gfCNCPoint5[13257] = {X 214.8514, Y 66.0622, Z -7.1667, A 0.000, B 0.000, C 0.000 }
gfCNCPoint5[13258] = {X 213.6675, Y 65.7094, Z -7.1667, A 0.000, B 0.000, C 0.000 }
gfCNCPoint5[13259] = {X 212.5602, Y 65.1615, Z -7.1667, A 0.000, B 0.000, C 0.000 }
gfCNCPoint5[13260] = {X 211.5615, Y 64.4343, Z -7.1667, A 0.000, B 0.000, C 0.000 }
gfCNCPoint5[13261] = {X 210.7002, Y 63.5486, Z -7.1667, A 0.000, B 0.000, C 0.000 }
gfCNCPoint5[13262] = {X 210.0010, Y 62.5301, Z -7.1667, A 0.000, B 0.000, C 0.000 }
gfCNCPoint5[13263] = {X 209.4841, Y 61.4080, Z -7.1667, A 0.000, B 0.000, C 0.000 }
gfCNCPoint5[13264] = {X 209.1643, Y 60.2147, Z -7.1667, A 0.000, B 0.000, C 0.000 }
gfCNCPoint5[13265] = {X 209.0510, Y 58.9845, Z -7.1667, A 0.000, B 0.000, C 0.000 }
gfCNCPoint5[13266] = {X 209.0508, Y 58.0000, Z -7.1667, A 0.000, B 0.000, C 0.000 }
gfCNCPoint5[13267] = {X 209.1477, Y 56.8162, Z -7.1667, A 0.000, B 0.000, C 0.000 }
gfCNCPoint5[13268] = {X 209.4358, Y 55.6638, Z -7.1667, A 0.000, B 0.000, C 0.000 }
gfCNCPoint5[13269] = {X 209.9075, Y 54.5737, Z -7.1667, A 0.000, B 0.000, C 0.000 }
gfCNCPoint5[13270] = {X 210.5502, Y 53.5748, Z -7.1667, A 0.000, B 0.000, C 0.000 }
gfCNCPoint5[13271] = {X 211.3467, Y 52.6937, Z -7.1667, A 0.000, B 0.000, C 0.000 }
gfCNCPoint5[13272] = {X 212.2759, Y 51.9538, Z -7.1667, A 0.000, B 0.000, C 0.000 }
gfCNCPoint5[13273] = {X 213.3131, Y 51.3749, Z -7.1667, A 0.000, B 0.000, C 0.000 }
gfCNCPoint5[13274] = {X 214.4306, Y 50.9724, Z -7.1667, A 0.000, B 0.000, C 0.000 }
gfCNCPoint5[13275] = {X 215.3724, Y 50.7834, Z -7.1667, A 0.000, B 0.000, C 0.000 }
gfCNCPoint5[13276] = {X 216.3308, Y 50.7200, Z -7.1667, A 0.000, B 0.000, C 0.000 }
gfCNCPoint5[13277] = {X 237.2617, Y 50.7200, Z -7.1667, A 0.000, B 0.000, C 0.000 }
gfCNCPoint5[13278] = {X 238.3057, Y 50.7953, Z -7.1667, A 0.000, B 0.000, C 0.000 }
gfCNCPoint5[13279] = {X 239.3282, Y 51.0195, Z -7.1667, A 0.000, B 0.000, C 0.000 }
gfCNCPoint5[13280] = {X 240.3080, Y 51.3880, Z -7.1667, A 0.000, B 0.000, C 0.000 }
gfCNCPoint5[13281] = {X 241.2247, Y 51.8932, Z -7.1667, A 0.000, B 0.000, C 0.000 }
gfCNCPoint5[13282] = {X 242.0740, Y 52.5374, Z -7.1667, A 0.000, B 0.000, C 0.000 }
gfCNCPoint5[13283] = {X 242.8201, Y 53.2987, Z -7.1667, A 0.000, B 0.000, C 0.000 }
gfCNCPoint5[13284] = {X 243.4471, Y 54.1608, Z -7.1667, A 0.000, B 0.000, C 0.000 }
gfCNCPoint5[13285] = {X 243.9414, Y 55.1053, Z -7.1667, A 0.000, B 0.000, C 0.000 }
gfCNCPoint5[13286] = {X 244.2925, Y 56.1117, Z -7.1667, A 0.000, B 0.000, C 0.000 }
gfCNCPoint5[13287] = {X 249.2045, Y 58.0272, Z -7.1667, A 0.000, B 0.000, C 0.000 }
gfCNCPoint5[13288] = {X 272.6717, Y 67.3417, Z -7.1667, A 0.000, B 0.000, C 0.000 }
gfCNCPoint5[13289] = {X 272.6716, Y 65.2836, Z -7.1667, A 0.000, B 0.000, C 0.000 }
gfCNCPoint5[13290] = {X 271.6643, Y 64.6022, Z -7.1667, A 0.000, B 0.000, C 0.000 }
gfCNCPoint5[13291] = {X 270.7845, Y 63.7626, Z -7.1667, A 0.000, B 0.000, C 0.000 }
gfCNCPoint5[13292] = {X 270.0567, Y 62.7883, Z -7.1667, A 0.000, B 0.000, C 0.000 }
gfCNCPoint5[13293] = {X 269.5012, Y 61.7064, Z -7.1667, A 0.000, B 0.000, C 0.000 }
gfCNCPoint5[13294] = {X 269.2026, Y 60.8250, Z -7.1667, A 0.000, B 0.000, C 0.000 }
gfCNCPoint5[13295] = {X 269.0188, Y 59.9127, Z -7.1667, A 0.000, B 0.000, C 0.000 }
gfCNCPoint5[13296] = {X 268.9529, Y 58.9845, Z -7.1667, A 0.000, B 0.000, C 0.000 }
gfCNCPoint5[13297] = {X 268.9527, Y 58.0000, Z -7.1667, A 0.000, B 0.000, C 0.000 }
gfCNCPoint5[13298] = {X 269.0633, Y 56.7358, Z -7.1667, A 0.000, B 0.000, C 0.000 }
gfCNCPoint5[13299] = {X 269.3917, Y 55.5101, Z -7.1667, A 0.000, B 0.000, C 0.000 }
gfCNCPoint5[13300] = {X 269.9280, Y 54.3600, Z -7.1667, A 0.000, B 0.000, C 0.000 }
gfCNCPoint5[13301] = {X 270.6559, Y 53.3205, Z -7.1667, A 0.000, B 0.000, C 0.000 }
gfCNCPoint5[13302] = {X 271.5532, Y 52.4232, Z -7.1667, A 0.000, B 0.000, C 0.000 }
gfCNCPoint5[13303] = {X 272.5927, Y 51.6953, Z -7.1667, A 0.000, B 0.000, C 0.000 }
gfCNCPoint5[13304] = {X 273.7428, Y 51.1590, Z -7.1667, A 0.000, B 0.000, C 0.000 }
gfCNCPoint5[13305] = {X 274.9685, Y 50.8306, Z -7.1667, A 0.000, B 0.000, C 0.000 }
gfCNCPoint5[13306] = {X 276.2327, Y 50.7200, Z -7.1667, A 0.000, B 0.000, C 0.000 }
gfCNCPoint5[13307] = {X 292.7731, Y 50.7200, Z -7.1667, A 0.000, B 0.000, C 0.000 }
gfCNCPoint5[13308] = {X 293.4209, Y 50.7489, Z -7.1667, A 0.000, B 0.000, C 0.000 }
gfCNCPoint5[13309] = {X 294.0636, Y 50.8353, Z -7.1667, A 0.000, B 0.000, C 0.000 }
gfCNCPoint5[13310] = {X 294.7292, Y 50.9877, Z -7.1667, A 0.000, B 0.000, C 0.000 }
gfCNCPoint5[13311] = {X 295.3777, Y 51.2019, Z -7.1667, A 0.000, B 0.000, C 0.000 }
gfCNCPoint5[13312] = {X 298.3089, Y 43.5511, Z -7.1667, A 0.000, B 0.000, C 0.000 }
gfCNCPoint5[13313] = {X 298.4820, Y 42.5283, Z -7.1667, A 0.000, B 0.000, C 0.000 }
gfCNCPoint5[13314] = {X 298.7923, Y 41.5385, Z -7.1667, A 0.000, B 0.000, C 0.000 }
gfCNCPoint5[13315] = {X 299.2339, Y 40.5998, Z -7.1667, A 0.000, B 0.000, C 0.000 }
gfCNCPoint5[13316] = {X 299.7987, Y 39.7298, Z -7.1667, A 0.000, B 0.000, C 0.000 }
gfCNCPoint5[13317] = {X 299.7987, Y 36.9943, Z -7.1667, A 0.000, B 0.000, C 0.000 }
gfCNCPoint5[13318] = {X 296.8149, Y 36.9943, Z -7.1667, A 0.000, B 0.000, C 0.000 }
gfCNCPoint5[13319] = {X 296.8147, Y 39.7480, Z -7.1667, A 0.000, B 0.000, C 0.000 }
gfCNCPoint5[13320] = {X 297.3857, Y 40.6103, Z -7.1667, A 0.000, B 0.000, C 0.000 }
gfCNCPoint5[13321] = {X 297.8305, Y 41.5440, Z -7.1667, A 0.000, B 0.000, C 0.000 }
gfCNCPoint5[13322] = {X 298.1402, Y 42.5307, Z -7.1667, A 0.000, B 0.000, C 0.000 }
gfCNCPoint5[13323] = {X 298.3089, Y 43.5511, Z -7.1667, A 0.000, B 0.000, C 0.000 }
gfCNCPoint5[13324] = {X 296.2363, Y 48.9607, Z -7.1667, A 0.000, B 0.000, C 0.000 }
gfCNCPoint5[13325] = {X 296.6124, Y 49.1139, Z -7.1667, A 0.000, B 0.000, C 0.000 }
gfCNCPoint5[13326] = {X 296.9817, Y 49.2828, Z -7.1667, A 0.000, B 0.000, C 0.000 }
gfCNCPoint5[13327] = {X 297.2571, Y 49.4212, Z -7.1667, A 0.000, B 0.000, C 0.000 }
gfCNCPoint5[13328] = {X 297.5280, Y 49.5683, Z -7.1667, A 0.000, B 0.000, C 0.000 }
gfCNCPoint5[13329] = {X 298.7174, Y 50.3602, Z -7.1667, A 0.000, B 0.000, C 0.000 }
gfCNCPoint5[13330] = {X 299.7774, Y 51.3185, Z -7.1667, A 0.000, B 0.000, C 0.000 }
gfCNCPoint5[13331] = {X 300.6847, Y 52.4224, Z -7.1667, A 0.000, B 0.000, C 0.000 }
gfCNCPoint5[13332] = {X 301.5914, Y 51.3191, Z -7.1667, A 0.000, B 0.000, C 0.000 }
gfCNCPoint5[13333] = {X 302.6506, Y 50.3611, Z -7.1667, A 0.000, B 0.000, C 0.000 }
gfCNCPoint5[13334] = {X 303.8393, Y 49.5695, Z -7.1667, A 0.000, B 0.000, C 0.000 }
gfCNCPoint5[13335] = {X 302.8989, Y 49.0956, Z -7.1667, A 0.000, B 0.000, C 0.000 }
gfCNCPoint5[13336] = {X 302.0820, Y 48.4310, Z -7.1667, A 0.000, B 0.000, C 0.000 }
gfCNCPoint5[13337] = {X 301.4268, Y 47.6067, Z -7.1667, A 0.000, B 0.000, C 0.000 }
gfCNCPoint5[13338] = {X 300.9636, Y 46.6610, Z -7.1667, A 0.000, B 0.000, C 0.000 }
gfCNCPoint5[13339] = {X 300.7923, Y 46.0759, Z -7.1667, A 0.000, B 0.000, C 0.000 }
gfCNCPoint5[13340] = {X 300.6953, Y 45.4741, Z -7.1667, A 0.000, B 0.000, C 0.000 }
gfCNCPoint5[13341] = {X 300.6790, Y 45.2570, Z -7.1667, A 0.000, B 0.000, C 0.000 }
gfCNCPoint5[13342] = {X 300.6724, Y 45.0393, Z -7.1667, A 0.000, B 0.000, C 0.000 }
gfCNCPoint5[13343] = {X 300.6725, Y 44.1884, Z -7.1667, A 0.000, B 0.000, C 0.000 }
gfCNCPoint5[13344] = {X 300.6810, Y 43.9888, Z -7.1667, A 0.000, B 0.000, C 0.000 }
gfCNCPoint5[13345] = {X 300.6970, Y 43.7898, Z -7.1667, A 0.000, B 0.000, C 0.000 }
gfCNCPoint5[13346] = {X 300.8617, Y 42.9110, Z -7.1667, A 0.000, B 0.000, C 0.000 }
gfCNCPoint5[13347] = {X 301.1736, Y 42.0731, Z -7.1667, A 0.000, B 0.000, C 0.000 }
gfCNCPoint5[13348] = {X 301.6237, Y 41.3006, Z -7.1667, A 0.000, B 0.000, C 0.000 }
gfCNCPoint5[13349] = {X 302.1987, Y 40.6160, Z -7.1667, A 0.000, B 0.000, C 0.000 }
gfCNCPoint5[13350] = {X 302.1987, Y 34.5943, Z -7.1667, A 0.000, B 0.000, C 0.000 }
gfCNCPoint5[13351] = {X 294.4151, Y 34.5943, Z -7.1667, A 0.000, B 0.000, C 0.000 }
gfCNCPoint5[13352] = {X 294.4146, Y 40.6550, Z -7.1667, A 0.000, B 0.000, C 0.000 }
gfCNCPoint5[13353] = {X 294.9946, Y 41.3214, Z -7.1667, A 0.000, B 0.000, C 0.000 }
gfCNCPoint5[13354] = {X 295.4475, Y 42.0800, Z -7.1667, A 0.000, B 0.000, C 0.000 }
gfCNCPoint5[13355] = {X 295.7590, Y 42.9067, Z -7.1667, A 0.000, B 0.000, C 0.000 }
gfCNCPoint5[13356] = {X 295.9194, Y 43.7755, Z -7.1667, A 0.000, B 0.000, C 0.000 }
gfCNCPoint5[13357] = {X 295.9350, Y 43.9919, Z -7.1667, A 0.000, B 0.000, C 0.000 }
gfCNCPoint5[13358] = {X 295.9411, Y 44.2089, Z -7.1667, A 0.000, B 0.000, C 0.000 }
gfCNCPoint5[13359] = {X 295.9411, Y 45.0000, Z -7.1667, A 0.000, B 0.000, C 0.000 }
gfCNCPoint5[13360] = {X 295.9354, Y 45.2373, Z -7.1667, A 0.000, B 0.000, C 0.000 }
gfCNCPoint5[13361] = {X 295.9181, Y 45.4741, Z -7.1667, A 0.000, B 0.000, C 0.000 }
gfCNCPoint5[13362] = {X 298.3067, Y 45.7073, Z -7.1667, A 0.000, B 0.000, C 0.000 }
gfCNCPoint5[13363] = {X 298.2010, Y 46.4214, Z -7.1667, A 0.000, B 0.000, C 0.000 }
gfCNCPoint5[13364] = {X 298.0252, Y 47.1215, Z -7.1667, A 0.000, B 0.000, C 0.000 }
gfCNCPoint5[13365] = {X 298.3689, Y 47.2942, Z -7.1667, A 0.000, B 0.000, C 0.000 }
gfCNCPoint5[13366] = {X 298.7069, Y 47.4778, Z -7.1667, A 0.000, B 0.000, C 0.000 }
gfCNCPoint5[13367] = {X 298.4514, Y 46.6051, Z -7.1667, A 0.000, B 0.000, C 0.000 }
gfCNCPoint5[13368] = {X 298.3067, Y 45.7073, Z -7.1667, A 0.000, B 0.000, C 0.000 }
gfCNCPoint5[13369] = {X 295.9181, Y 45.4741, Z -7.1667, A 0.000, B 0.000, C 0.000 }
gfCNCPoint5[13370] = {X 295.8472, Y 45.9528, Z -7.1667, A 0.000, B 0.000, C 0.000 }
gfCNCPoint5[13371] = {X 295.7293, Y 46.4221, Z -7.1667, A 0.000, B 0.000, C 0.000 }
gfCNCPoint5[13372] = {X 295.4314, Y 47.1714, Z -7.1667, A 0.000, B 0.000, C 0.000 }
gfCNCPoint5[13373] = {X 295.0142, Y 47.8614, Z -7.1667, A 0.000, B 0.000, C 0.000 }
gfCNCPoint5[13374] = {X 294.4890, Y 48.4733, Z -7.1667, A 0.000, B 0.000, C 0.000 }
gfCNCPoint5[13375] = {X 295.3741, Y 48.6760, Z -7.1667, A 0.000, B 0.000, C 0.000 }
gfCNCPoint5[13376] = {X 296.2363, Y 48.9607, Z -7.1667, A 0.000, B 0.000, C 0.000 }
gfCNCPoint5[13377] = {X 295.3777, Y 51.2019, Z -7.1667, A 0.000, B 0.000, C 0.000 }
gfCNCPoint5[13378] = {X 296.3498, Y 51.6592, Z -7.1667, A 0.000, B 0.000, C 0.000 }
gfCNCPoint5[13379] = {X 297.2441, Y 52.2547, Z -7.1667, A 0.000, B 0.000, C 0.000 }
gfCNCPoint5[13380] = {X 298.0410, Y 52.9753, Z -7.1667, A 0.000, B 0.000, C 0.000 }
gfCNCPoint5[13381] = {X 298.7231, Y 53.8053, Z -7.1667, A 0.000, B 0.000, C 0.000 }
gfCNCPoint5[13382] = {X 299.2946, Y 54.7645, Z -7.1667, A 0.000, B 0.000, C 0.000 }
gfCNCPoint5[13383] = {X 299.7126, Y 55.7997, Z -7.1667, A 0.000, B 0.000, C 0.000 }
gfCNCPoint5[13384] = {X 299.9675, Y 56.8868, Z -7.1667, A 0.000, B 0.000, C 0.000 }
gfCNCPoint5[13385] = {X 300.0531, Y 58.0000, Z -7.1667, A 0.000, B 0.000, C 0.000 }
gfCNCPoint5[13386] = {X 300.0531, Y 58.9431, Z -7.1667, A 0.000, B 0.000, C 0.000 }
gfCNCPoint5[13387] = {X 299.9650, Y 60.0533, Z -7.1667, A 0.000, B 0.000, C 0.000 }
gfCNCPoint5[13388] = {X 299.7090, Y 61.1372, Z -7.1667, A 0.000, B 0.000, C 0.000 }
gfCNCPoint5[13389] = {X 299.2910, Y 62.1695, Z -7.1667, A 0.000, B 0.000, C 0.000 }
gfCNCPoint5[13390] = {X 298.7208, Y 63.1261, Z -7.1667, A 0.000, B 0.000, C 0.000 }
gfCNCPoint5[13391] = {X 300.6826, Y 64.5087, Z -7.1667, A 0.000, B 0.000, C 0.000 }
gfCNCPoint5[13392] = {X 299.7833, Y 65.6047, Z -7.1667, A 0.000, B 0.000, C 0.000 }
gfCNCPoint5[13393] = {X 298.7338, Y 66.5579, Z -7.1667, A 0.000, B 0.000, C 0.000 }
gfCNCPoint5[13394] = {X 298.7338, Y 89.4417, Z -7.1667, A 0.000, B 0.000, C 0.000 }
gfCNCPoint5[13395] = {X 299.8304, Y 90.4463, Z -7.1667, A 0.000, B 0.000, C 0.000 }
gfCNCPoint5[13396] = {X 300.7607, Y 91.6065, Z -7.1667, A 0.000, B 0.000, C 0.000 }
gfCNCPoint5[13397] = {X 301.5031, Y 92.8951, Z -7.1667, A 0.000, B 0.000, C 0.000 }
gfCNCPoint5[13398] = {X 304.0666, Y 92.8951, Z -7.1667, A 0.000, B 0.000, C 0.000 }
gfCNCPoint5[13399] = {X 303.7091, Y 91.9009, Z -7.1667, A 0.000, B 0.000, C 0.000 }
gfCNCPoint5[13400] = {X 303.4130, Y 90.8868, Z -7.1667, A 0.000, B 0.000, C 0.000 }
gfCNCPoint5[13401] = {X 302.9737, Y 88.8157, Z -7.1667, A 0.000, B 0.000, C 0.000 }
gfCNCPoint5[13402] = {X 302.7135, Y 86.7145, Z -7.1667, A 0.000, B 0.000, C 0.000 }
gfCNCPoint5[13403] = {X 302.6344, Y 84.5988, Z -7.1667, A 0.000, B 0.000, C 0.000 }
gfCNCPoint5[13404] = {X 302.6354, Y 66.5611, Z -7.1667, A 0.000, B 0.000, C 0.000 }
gfCNCPoint5[13405] = {X 301.5835, Y 65.6067, Z -7.1667, A 0.000, B 0.000, C 0.000 }
gfCNCPoint5[13406] = {X 300.6826, Y 64.5087, Z -7.1667, A 0.000, B 0.000, C 0.000 }
gfCNCPoint5[13407] = {X 298.7208, Y 63.1261, Z -7.1667, A 0.000, B 0.000, C 0.000 }
gfCNCPoint5[13408] = {X 298.0349, Y 63.9605, Z -7.1667, A 0.000, B 0.000, C 0.000 }
gfCNCPoint5[13409] = {X 297.2334, Y 64.6845, Z -7.1667, A 0.000, B 0.000, C 0.000 }
gfCNCPoint5[13410] = {X 296.3338, Y 65.2822, Z -7.1667, A 0.000, B 0.000, C 0.000 }
gfCNCPoint5[13411] = {X 296.3338, Y 90.7159, Z -7.1667, A 0.000, B 0.000, C 0.000 }
gfCNCPoint5[13412] = {X 297.3139, Y 91.3787, Z -7.1667, A 0.000, B 0.000, C 0.000 }
gfCNCPoint5[13413] = {X 298.1742, Y 92.1909, Z -7.1667, A 0.000, B 0.000, C 0.000 }
gfCNCPoint5[13414] = {X 298.8923, Y 93.1313, Z -7.1667, A 0.000, B 0.000, C 0.000 }
gfCNCPoint5[13415] = {X 299.4494, Y 94.1751, Z -7.1667, A 0.000, B 0.000, C 0.000 }
gfCNCPoint5[13416] = {X 299.8308, Y 95.2951, Z -7.1667, A 0.000, B 0.000, C 0.000 }
gfCNCPoint5[13417] = {X 308.0988, Y 95.2951, Z -7.1667, A 0.000, B 0.000, C 0.000 }
gfCNCPoint5[13418] = {X 307.0955, Y 93.7115, Z -7.1667, A 0.000, B 0.000, C 0.000 }
gfCNCPoint5[13419] = {X 306.2992, Y 92.0144, Z -7.1667, A 0.000, B 0.000, C 0.000 }
gfCNCPoint5[13420] = {X 305.9913, Y 91.1582, Z -7.1667, A 0.000, B 0.000, C 0.000 }
gfCNCPoint5[13421] = {X 305.7363, Y 90.2848, Z -7.1667, A 0.000, B 0.000, C 0.000 }
gfCNCPoint5[13422] = {X 305.3399, Y 88.4142, Z -7.1667, A 0.000, B 0.000, C 0.000 }
gfCNCPoint5[13423] = {X 305.1053, Y 86.5166, Z -7.1667, A 0.000, B 0.000, C 0.000 }
gfCNCPoint5[13424] = {X 305.0344, Y 84.6058, Z -7.1667, A 0.000, B 0.000, C 0.000 }
gfCNCPoint5[13425] = {X 305.0355, Y 65.2838, Z -7.1667, A 0.000, B 0.000, C 0.000 }
gfCNCPoint5[13426] = {X 304.1342, Y 64.6863, Z -7.1667, A 0.000, B 0.000, C 0.000 }
gfCNCPoint5[13427] = {X 303.3313, Y 63.9619, Z -7.1667, A 0.000, B 0.000, C 0.000 }
gfCNCPoint5[13428] = {X 302.6446, Y 63.1265, Z -7.1667, A 0.000, B 0.000, C 0.000 }
gfCNCPoint5[13429] = {X 302.0794, Y 62.1790, Z -7.1667, A 0.000, B 0.000, C 0.000 }
gfCNCPoint5[13430] = {X 301.6639, Y 61.1570, Z -7.1667, A 0.000, B 0.000, C 0.000 }
gfCNCPoint5[13431] = {X 301.4076, Y 60.0840, Z -7.1667, A 0.000, B 0.000, C 0.000 }
gfCNCPoint5[13432] = {X 301.3164, Y 58.9845, Z -7.1667, A 0.000, B 0.000, C 0.000 }
gfCNCPoint5[13433] = {X 301.3162, Y 58.0000, Z -7.1667, A 0.000, B 0.000, C 0.000 }
gfCNCPoint5[13434] = {X 301.4018, Y 56.8868, Z -7.1667, A 0.000, B 0.000, C 0.000 }
gfCNCPoint5[13435] = {X 301.6567, Y 55.7997, Z -7.1667, A 0.000, B 0.000, C 0.000 }
gfCNCPoint5[13436] = {X 302.0747, Y 54.7645, Z -7.1667, A 0.000, B 0.000, C 0.000 }
gfCNCPoint5[13437] = {X 302.6462, Y 53.8053, Z -7.1667, A 0.000, B 0.000, C 0.000 }
gfCNCPoint5[13438] = {X 303.3281, Y 52.9755, Z -7.1667, A 0.000, B 0.000, C 0.000 }
gfCNCPoint5[13439] = {X 304.1247, Y 52.2551, Z -7.1667, A 0.000, B 0.000, C 0.000 }
gfCNCPoint5[13440] = {X 305.0187, Y 51.6597, Z -7.1667, A 0.000, B 0.000, C 0.000 }
gfCNCPoint5[13441] = {X 306.1514, Y 51.1428, Z -7.1667, A 0.000, B 0.000, C 0.000 }
gfCNCPoint5[13442] = {X 307.3557, Y 50.8265, Z -7.1667, A 0.000, B 0.000, C 0.000 }
gfCNCPoint5[13443] = {X 308.5962, Y 50.7200, Z -7.1667, A 0.000, B 0.000, C 0.000 }
gfCNCPoint5[13444] = {X 324.3107, Y 50.7200, Z -7.1667, A 0.000, B 0.000, C 0.000 }
gfCNCPoint5[13445] = {X 325.2469, Y 50.7804, Z -7.1667, A 0.000, B 0.000, C 0.000 }
gfCNCPoint5[13446] = {X 326.1675, Y 50.9608, Z -7.1667, A 0.000, B 0.000, C 0.000 }
gfCNCPoint5[13447] = {X 326.5260, Y 51.0653, Z -7.1667, A 0.000, B 0.000, C 0.000 }
gfCNCPoint5[13448] = {X 326.8787, Y 51.1880, Z -7.1667, A 0.000, B 0.000, C 0.000 }
gfCNCPoint5[13449] = {X 327.4507, Y 51.4320, Z -7.1667, A 0.000, B 0.000, C 0.000 }
gfCNCPoint5[13450] = {X 327.9997, Y 51.7239, Z -7.1667, A 0.000, B 0.000, C 0.000 }
gfCNCPoint5[13451] = {X 328.5431, Y 52.0767, Z -7.1667, A 0.000, B 0.000, C 0.000 }
gfCNCPoint5[13452] = {X 329.0529, Y 52.4765, Z -7.1667, A 0.000, B 0.000, C 0.000 }
gfCNCPoint5[13453] = {X 329.9296, Y 53.3711, Z -7.1667, A 0.000, B 0.000, C 0.000 }
gfCNCPoint5[13454] = {X 330.6399, Y 54.4029, Z -7.1667, A 0.000, B 0.000, C 0.000 }
gfCNCPoint5[13455] = {X 331.1628, Y 55.5411, Z -7.1667, A 0.000, B 0.000, C 0.000 }
gfCNCPoint5[13456] = {X 331.4829, Y 56.7521, Z -7.1667, A 0.000, B 0.000, C 0.000 }
gfCNCPoint5[13457] = {X 331.5907, Y 58.0000, Z -7.1667, A 0.000, B 0.000, C 0.000 }
gfCNCPoint5[13458] = {X 331.5907, Y 58.9393, Z -7.1667, A 0.000, B 0.000, C 0.000 }
gfCNCPoint5[13459] = {X 331.4737, Y 60.2164, Z -7.1667, A 0.000, B 0.000, C 0.000 }
gfCNCPoint5[13460] = {X 331.1355, Y 61.4535, Z -7.1667, A 0.000, B 0.000, C 0.000 }
gfCNCPoint5[13461] = {X 330.5865, Y 62.6125, Z -7.1667, A 0.000, B 0.000, C 0.000 }
gfCNCPoint5[13462] = {X 329.8436, Y 63.6579, Z -7.1667, A 0.000, B 0.000, C 0.000 }
gfCNCPoint5[13463] = {X 328.9296, Y 64.5576, Z -7.1667, A 0.000, B 0.000, C 0.000 }
gfCNCPoint5[13464] = {X 327.8725, Y 65.2838, Z -7.1667, A 0.000, B 0.000, C 0.000 }
gfCNCPoint5[13465] = {X 327.8742, Y 83.2150, Z -7.1667, A 0.000, B 0.000, C 0.000 }
gfCNCPoint5[13466] = {X 327.8877, Y 84.5911, Z -7.1667, A 0.000, B 0.000, C 0.000 }
gfCNCPoint5[13467] = {X 327.8972, Y 84.9519, Z -7.1667, A 0.000, B 0.000, C 0.000 }
gfCNCPoint5[13468] = {X 327.9238, Y 85.3118, Z -7.1667, A 0.000, B 0.000, C 0.000 }
gfCNCPoint5[13469] = {X 329.1610, Y 85.7652, Z -7.1667, A 0.000, B 0.000, C 0.000 }
gfCNCPoint5[13470] = {X 330.4377, Y 86.0909, Z -7.1667, A 0.000, B 0.000, C 0.000 }
gfCNCPoint5[13471] = {X 333.3490, Y 86.6140, Z -7.1667, A 0.000, B 0.000, C 0.000 }
gfCNCPoint5[13472] = {X 336.2868, Y 86.9583, Z -7.1667, A 0.000, B 0.000, C 0.000 }
gfCNCPoint5[13473] = {X 340.5661, Y 87.2462, Z -7.1667, A 0.000, B 0.000, C 0.000 }
gfCNCPoint5[13474] = {X 344.8525, Y 87.3965, Z -7.1667, A 0.000, B 0.000, C 0.000 }
gfCNCPoint5[13475] = {X 349.1414, Y 87.4090, Z -7.1667, A 0.000, B 0.000, C 0.000 }
gfCNCPoint5[13476] = {X 353.1932, Y 87.3432, Z -7.1667, A 0.000, B 0.000, C 0.000 }
gfCNCPoint5[13477] = {X 357.2400, Y 87.1300, Z -7.1667, A 0.000, B 0.000, C 0.000 }
gfCNCPoint5[13478] = {X 361.2763, Y 86.7697, Z -7.1667, A 0.000, B 0.000, C 0.000 }
gfCNCPoint5[13479] = {X 363.1974, Y 86.5045, Z -7.1667, A 0.000, B 0.000, C 0.000 }
gfCNCPoint5[13480] = {X 365.1009, Y 86.1330, Z -7.1667, A 0.000, B 0.000, C 0.000 }
gfCNCPoint5[13481] = {X 366.9808, Y 85.6565, Z -7.1667, A 0.000, B 0.000, C 0.000 }
gfCNCPoint5[13482] = {X 367.4412, Y 85.5106, Z -7.1667, A 0.000, B 0.000, C 0.000 }
gfCNCPoint5[13483] = {X 367.8879, Y 85.3265, Z -7.1667, A 0.000, B 0.000, C 0.000 }
gfCNCPoint5[13484] = {X 367.9413, Y 84.5786, Z -7.1667, A 0.000, B 0.000, C 0.000 }
gfCNCPoint5[13485] = {X 367.9591, Y 83.8290, Z -7.1667, A 0.000, B 0.000, C 0.000 }
gfCNCPoint5[13486] = {X 367.9580, Y 65.2835, Z -7.1667, A 0.000, B 0.000, C 0.000 }
gfCNCPoint5[13487] = {X 366.9044, Y 64.5644, Z -7.1667, A 0.000, B 0.000, C 0.000 }
gfCNCPoint5[13488] = {X 365.9924, Y 63.6724, Z -7.1667, A 0.000, B 0.000, C 0.000 }
gfCNCPoint5[13489] = {X 365.2502, Y 62.6349, Z -7.1667, A 0.000, B 0.000, C 0.000 }
gfCNCPoint5[13490] = {X 364.7004, Y 61.4838, Z -7.1667, A 0.000, B 0.000, C 0.000 }
gfCNCPoint5[13491] = {X 364.3600, Y 60.2544, Z -7.1667, A 0.000, B 0.000, C 0.000 }
gfCNCPoint5[13492] = {X 364.2395, Y 58.9845, Z -7.1667, A 0.000, B 0.000, C 0.000 }
gfCNCPoint5[13493] = {X 364.2393, Y 58.0000, Z -7.1667, A 0.000, B 0.000, C 0.000 }
gfCNCPoint5[13494] = {X 364.3499, Y 56.7358, Z -7.1667, A 0.000, B 0.000, C 0.000 }
gfCNCPoint5[13495] = {X 364.6783, Y 55.5101, Z -7.1667, A 0.000, B 0.000, C 0.000 }
gfCNCPoint5[13496] = {X 365.2146, Y 54.3600, Z -7.1667, A 0.000, B 0.000, C 0.000 }
gfCNCPoint5[13497] = {X 365.9425, Y 53.3205, Z -7.1667, A 0.000, B 0.000, C 0.000 }
gfCNCPoint5[13498] = {X 366.8398, Y 52.4232, Z -7.1667, A 0.000, B 0.000, C 0.000 }
gfCNCPoint5[13499] = {X 367.8793, Y 51.6953, Z -7.1667, A 0.000, B 0.000, C 0.000 }
gfCNCPoint5[13500] = {X 369.0294, Y 51.1590, Z -7.1667, A 0.000, B 0.000, C 0.000 }
gfCNCPoint5[13501] = {X 370.2551, Y 50.8306, Z -7.1667, A 0.000, B 0.000, C 0.000 }
gfCNCPoint5[13502] = {X 371.5193, Y 50.7200, Z -7.1667, A 0.000, B 0.000, C 0.000 }
gfCNCPoint5[13503] = {X 388.0597, Y 50.7200, Z -7.1667, A 0.000, B 0.000, C 0.000 }
gfCNCPoint5[13504] = {X 389.2271, Y 50.8142, Z -7.1667, A 0.000, B 0.000, C 0.000 }
gfCNCPoint5[13505] = {X 390.3643, Y 51.0944, Z -7.1667, A 0.000, B 0.000, C 0.000 }
gfCNCPoint5[13506] = {X 391.4418, Y 51.5533, Z -7.1667, A 0.000, B 0.000, C 0.000 }
gfCNCPoint5[13507] = {X 392.4319, Y 52.1791, Z -7.1667, A 0.000, B 0.000, C 0.000 }
gfCNCPoint5[13508] = {X 393.3087, Y 52.9556, Z -7.1667, A 0.000, B 0.000, C 0.000 }
gfCNCPoint5[13509] = {X 394.1855, Y 52.1791, Z -7.1667, A 0.000, B 0.000, C 0.000 }
gfCNCPoint5[13510] = {X 395.1756, Y 51.5533, Z -7.1667, A 0.000, B 0.000, C 0.000 }
gfCNCPoint5[13511] = {X 396.2531, Y 51.0944, Z -7.1667, A 0.000, B 0.000, C 0.000 }
gfCNCPoint5[13512] = {X 397.3903, Y 50.8142, Z -7.1667, A 0.000, B 0.000, C 0.000 }
gfCNCPoint5[13513] = {X 398.5577, Y 50.7200, Z -7.1667, A 0.000, B 0.000, C 0.000 }
gfCNCPoint5[13514] = {X 419.4886, Y 50.7200, Z -7.1667, A 0.000, B 0.000, C 0.000 }
gfCNCPoint5[13515] = {X 420.6739, Y 50.8171, Z -7.1667, A 0.000, B 0.000, C 0.000 }
gfCNCPoint5[13516] = {X 421.8275, Y 51.1059, Z -7.1667, A 0.000, B 0.000, C 0.000 }
gfCNCPoint5[13517] = {X 422.9187, Y 51.5787, Z -7.1667, A 0.000, B 0.000, C 0.000 }
gfCNCPoint5[13518] = {X 423.9184, Y 52.2228, Z -7.1667, A 0.000, B 0.000, C 0.000 }
gfCNCPoint5[13519] = {X 424.7998, Y 53.0211, Z -7.1667, A 0.000, B 0.000, C 0.000 }
gfCNCPoint5[13520] = {X 425.5396, Y 53.9523, Z -7.1667, A 0.000, B 0.000, C 0.000 }
gfCNCPoint5[13521] = {X 426.1179, Y 54.9914, Z -7.1667, A 0.000, B 0.000, C 0.000 }
gfCNCPoint5[13522] = {X 426.5192, Y 56.1109, Z -7.1667, A 0.000, B 0.000, C 0.000 }
gfCNCPoint5[13523] = {X 430.7006, Y 57.7400, Z -7.1667, A 0.000, B 0.000, C 0.000 }
gfCNCPoint5[13524] = {X 454.8981, Y 67.3409, Z -7.1667, A 0.000, B 0.000, C 0.000 }
gfCNCPoint5[13525] = {X 454.8982, Y 65.2835, Z -7.1667, A 0.000, B 0.000, C 0.000 }
gfCNCPoint5[13526] = {X 453.8910, Y 64.6021, Z -7.1667, A 0.000, B 0.000, C 0.000 }
gfCNCPoint5[13527] = {X 453.0113, Y 63.7626, Z -7.1667, A 0.000, B 0.000, C 0.000 }
gfCNCPoint5[13528] = {X 452.2836, Y 62.7884, Z -7.1667, A 0.000, B 0.000, C 0.000 }
gfCNCPoint5[13529] = {X 451.7282, Y 61.7066, Z -7.1667, A 0.000, B 0.000, C 0.000 }
gfCNCPoint5[13530] = {X 451.4295, Y 60.8252, Z -7.1667, A 0.000, B 0.000, C 0.000 }
gfCNCPoint5[13531] = {X 451.2457, Y 59.9128, Z -7.1667, A 0.000, B 0.000, C 0.000 }
gfCNCPoint5[13532] = {X 451.1798, Y 58.9845, Z -7.1667, A 0.000, B 0.000, C 0.000 }
gfCNCPoint5[13533] = {X 451.1796, Y 58.0000, Z -7.1667, A 0.000, B 0.000, C 0.000 }
gfCNCPoint5[13534] = {X 451.2795, Y 56.7981, Z -7.1667, A 0.000, B 0.000, C 0.000 }
gfCNCPoint5[13535] = {X 451.5765, Y 55.6291, Z -7.1667, A 0.000, B 0.000, C 0.000 }
gfCNCPoint5[13536] = {X 452.0624, Y 54.5253, Z -7.1667, A 0.000, B 0.000, C 0.000 }
gfCNCPoint5[13537] = {X 452.7238, Y 53.5168, Z -7.1667, A 0.000, B 0.000, C 0.000 }
gfCNCPoint5[13538] = {X 453.5427, Y 52.6313, Z -7.1667, A 0.000, B 0.000, C 0.000 }
gfCNCPoint5[13539] = {X 454.4966, Y 51.8932, Z -7.1667, A 0.000, B 0.000, C 0.000 }
gfCNCPoint5[13540] = {X 455.4133, Y 51.3880, Z -7.1667, A 0.000, B 0.000, C 0.000 }
gfCNCPoint5[13541] = {X 456.3931, Y 51.0195, Z -7.1667, A 0.000, B 0.000, C 0.000 }
gfCNCPoint5[13542] = {X 457.4155, Y 50.7953, Z -7.1667, A 0.000, B 0.000, C 0.000 }
gfCNCPoint5[13543] = {X 458.4596, Y 50.7200, Z -7.1667, A 0.000, B 0.000, C 0.000 }
gfCNCPoint5[13544] = {X 475.0000, Y 50.7200, Z -7.1667, A 0.000, B 0.000, C 0.000 }
gfCNCPoint5[13545] = {X 476.0441, Y 50.7953, Z -7.1667, A 0.000, B 0.000, C 0.000 }
gfCNCPoint5[13546] = {X 477.0665, Y 51.0195, Z -7.1667, A 0.000, B 0.000, C 0.000 }
gfCNCPoint5[13547] = {X 478.0463, Y 51.3880, Z -7.1667, A 0.000, B 0.000, C 0.000 }
gfCNCPoint5[13548] = {X 478.9630, Y 51.8932, Z -7.1667, A 0.000, B 0.000, C 0.000 }
gfCNCPoint5[13549] = {X 479.9169, Y 52.6313, Z -7.1667, A 0.000, B 0.000, C 0.000 }
gfCNCPoint5[13550] = {X 480.7358, Y 53.5168, Z -7.1667, A 0.000, B 0.000, C 0.000 }
gfCNCPoint5[13551] = {X 481.3972, Y 54.5253, Z -7.1667, A 0.000, B 0.000, C 0.000 }
gfCNCPoint5[13552] = {X 481.8831, Y 55.6291, Z -7.1667, A 0.000, B 0.000, C 0.000 }
gfCNCPoint5[13553] = {X 482.1801, Y 56.7981, Z -7.1667, A 0.000, B 0.000, C 0.000 }
gfCNCPoint5[13554] = {X 482.2800, Y 58.0000, Z -7.1667, A 0.000, B 0.000, C 0.000 }
gfCNCPoint5[13555] = {X 482.2798, Y 58.9942, Z -7.1667, A 0.000, B 0.000, C 0.000 }
gfCNCPoint5[13556] = {X 482.1578, Y 60.2625, Z -7.1667, A 0.000, B 0.000, C 0.000 }
gfCNCPoint5[13557] = {X 481.8166, Y 61.4900, Z -7.1667, A 0.000, B 0.000, C 0.000 }
gfCNCPoint5[13558] = {X 481.2666, Y 62.6393, Z -7.1667, A 0.000, B 0.000, C 0.000 }
gfCNCPoint5[13559] = {X 480.5246, Y 63.6750, Z -7.1667, A 0.000, B 0.000, C 0.000 }
gfCNCPoint5[13560] = {X 479.6135, Y 64.5656, Z -7.1667, A 0.000, B 0.000, C 0.000 }
gfCNCPoint5[13561] = {X 478.5610, Y 65.2837, Z -7.1667, A 0.000, B 0.000, C 0.000 }
gfCNCPoint5[13562] = {X 478.5614, Y 90.7244, Z -7.1667, A 0.000, B 0.000, C 0.000 }
gfCNCPoint5[13563] = {X 479.5435, Y 91.3834, Z -7.1667, A 0.000, B 0.000, C 0.000 }
gfCNCPoint5[13564] = {X 480.4055, Y 92.1931, Z -7.1667, A 0.000, B 0.000, C 0.000 }
gfCNCPoint5[13565] = {X 481.1246, Y 93.1320, Z -7.1667, A 0.000, B 0.000, C 0.000 }
gfCNCPoint5[13566] = {X 481.6816, Y 94.1753, Z -7.1667, A 0.000, B 0.000, C 0.000 }
gfCNCPoint5[13567] = {X 482.0619, Y 95.2951, Z -7.1667, A 0.000, B 0.000, C 0.000 }
gfCNCPoint5[13568] = {X 507.6812, Y 95.2951, Z -7.1667, A 0.000, B 0.000, C 0.000 }
gfCNCPoint5[13569] = {X 507.6812, Y 97.6951, Z -7.1667, A 0.000, B 0.000, C 0.000 }
gfCNCPoint5[13570] = {X 597.6967, Y 97.6951, Z -7.1667, A 0.000, B 0.000, C 0.000 }
gfCNCPoint5[13571] = {X 597.6967, Y 51.8000, Z -7.1667, A 0.000, B 0.000, C 0.000 }
gfCNCPoint5[13572] = {X 593.5565, Y 51.8000, Z -7.1667, A 0.000, B 0.000, C 0.000 }
gfCNCPoint5[13573] = {X 592.3428, Y 51.6908, Z -7.1667, A 0.000, B 0.000, C 0.000 }
gfCNCPoint5[13574] = {X 591.1680, Y 51.3667, Z -7.1667, A 0.000, B 0.000, C 0.000 }
gfCNCPoint5[13575] = {X 590.0699, Y 50.8381, Z -7.1667, A 0.000, B 0.000, C 0.000 }
gfCNCPoint5[13576] = {X 589.0838, Y 50.1220, Z -7.1667, A 0.000, B 0.000, C 0.000 }
gfCNCPoint5[13577] = {X 588.4736, Y 49.5171, Z -7.1667, A 0.000, B 0.000, C 0.000 }
gfCNCPoint5[13578] = {X 587.9446, Y 48.8401, Z -7.1667, A 0.000, B 0.000, C 0.000 }
gfCNCPoint5[13579] = {X 587.5052, Y 48.1018, Z -7.1667, A 0.000, B 0.000, C 0.000 }
gfCNCPoint5[13580] = {X 587.0658, Y 48.8401, Z -7.1667, A 0.000, B 0.000, C 0.000 }
gfCNCPoint5[13581] = {X 586.5368, Y 49.5171, Z -7.1667, A 0.000, B 0.000, C 0.000 }
gfCNCPoint5[13582] = {X 585.9266, Y 50.1220, Z -7.1667, A 0.000, B 0.000, C 0.000 }
gfCNCPoint5[13583] = {X 585.1803, Y 50.6880, Z -7.1667, A 0.000, B 0.000, C 0.000 }
gfCNCPoint5[13584] = {X 584.3634, Y 51.1461, Z -7.1667, A 0.000, B 0.000, C 0.000 }
gfCNCPoint5[13585] = {X 583.3013, Y 51.5442, Z -7.1667, A 0.000, B 0.000, C 0.000 }
gfCNCPoint5[13586] = {X 582.1877, Y 51.7603, Z -7.1667, A 0.000, B 0.000, C 0.000 }
gfCNCPoint5[13587] = {X 581.0538, Y 51.7882, Z -7.1667, A 0.000, B 0.000, C 0.000 }
gfCNCPoint5[13588] = {X 579.9310, Y 51.6273, Z -7.1667, A 0.000, B 0.000, C 0.000 }
gfCNCPoint5[13589] = {X 578.8505, Y 51.2819, Z -7.1667, A 0.000, B 0.000, C 0.000 }
gfCNCPoint5[13590] = {X 577.8425, Y 50.7618, Z -7.1667, A 0.000, B 0.000, C 0.000 }
gfCNCPoint5[13591] = {X 576.9350, Y 50.0813, Z -7.1667, A 0.000, B 0.000, C 0.000 }
gfCNCPoint5[13592] = {X 576.3133, Y 49.4513, Z -7.1667, A 0.000, B 0.000, C 0.000 }
gfCNCPoint5[13593] = {X 575.7786, Y 48.7459, Z -7.1667, A 0.000, B 0.000, C 0.000 }
gfCNCPoint5[13594] = {X 575.3401, Y 47.9770, Z -7.1667, A 0.000, B 0.000, C 0.000 }
gfCNCPoint5[13595] = {X 574.9017, Y 48.7459, Z -7.1667, A 0.000, B 0.000, C 0.000 }
gfCNCPoint5[13596] = {X 574.3670, Y 49.4513, Z -7.1667, A 0.000, B 0.000, C 0.000 }
gfCNCPoint5[13597] = {X 573.7453, Y 50.0813, Z -7.1667, A 0.000, B 0.000, C 0.000 }
gfCNCPoint5[13598] = {X 572.7526, Y 50.8143, Z -7.1667, A 0.000, B 0.000, C 0.000 }
gfCNCPoint5[13599] = {X 571.6437, Y 51.3558, Z -7.1667, A 0.000, B 0.000, C 0.000 }
gfCNCPoint5[13600] = {X 570.4553, Y 51.6880, Z -7.1667, A 0.000, B 0.000, C 0.000 }
gfCNCPoint5[13601] = {X 569.2264, Y 51.8000, Z -7.1667, A 0.000, B 0.000, C 0.000 }
gfCNCPoint5[13602] = {X 562.4443, Y 51.8000, Z -7.1667, A 0.000, B 0.000, C 0.000 }
gfCNCPoint5[13603] = {X 561.3805, Y 51.7163, Z -7.1667, A 0.000, B 0.000, C 0.000 }
gfCNCPoint5[13604] = {X 560.3430, Y 51.4672, Z -7.1667, A 0.000, B 0.000, C 0.000 }
gfCNCPoint5[13605] = {X 559.3572, Y 51.0588, Z -7.1667, A 0.000, B 0.000, C 0.000 }
gfCNCPoint5[13606] = {X 558.4474, Y 50.5013, Z -7.1667, A 0.000, B 0.000, C 0.000 }
gfCNCPoint5[13607] = {X 557.6360, Y 49.8083, Z -7.1667, A 0.000, B 0.000, C 0.000 }
gfCNCPoint5[13608] = {X 556.9430, Y 48.9969, Z -7.1667, A 0.000, B 0.000, C 0.000 }
gfCNCPoint5[13609] = {X 556.3855, Y 48.0871, Z -7.1667, A 0.000, B 0.000, C 0.000 }
gfCNCPoint5[13610] = {X 555.9771, Y 47.1013, Z -7.1667, A 0.000, B 0.000, C 0.000 }
gfCNCPoint5[13611] = {X 555.7280, Y 46.0638, Z -7.1667, A 0.000, B 0.000, C 0.000 }
gfCNCPoint5[13612] = {X 555.6443, Y 45.0000, Z -7.1667, A 0.000, B 0.000, C 0.000 }
gfCNCPoint5[13613] = {X 555.6443, Y 44.0565, Z -7.1667, A 0.000, B 0.000, C 0.000 }
gfCNCPoint5[13614] = {X 555.7462, Y 42.9041, Z -7.1667, A 0.000, B 0.000, C 0.000 }
gfCNCPoint5[13615] = {X 556.0411, Y 41.7855, Z -7.1667, A 0.000, B 0.000, C 0.000 }
gfCNCPoint5[13616] = {X 556.5206, Y 40.7326, Z -7.1667, A 0.000, B 0.000, C 0.000 }
gfCNCPoint5[13617] = {X 557.1709, Y 39.7758, Z -7.1667, A 0.000, B 0.000, C 0.000 }
gfCNCPoint5[13618] = {X 557.1710, Y 10.2274, Z -7.1667, A 0.000, B 0.000, C 0.000 }
gfCNCPoint5[13619] = {X 556.5252, Y 9.2814, Z -7.1667, A 0.000, B 0.000, C 0.000 }
gfCNCPoint5[13620] = {X 556.0474, Y 8.2404, Z -7.1667, A 0.000, B 0.000, C 0.000 }
gfCNCPoint5[13621] = {X 555.7510, Y 7.1340, Z -7.1667, A 0.000, B 0.000, C 0.000 }
gfCNCPoint5[13622] = {X 555.6446, Y 5.9935, Z -7.1667, A 0.000, B 0.000, C 0.000 }
gfCNCPoint5[13623] = {X 555.6443, Y 5.0000, Z -7.1667, A 0.000, B 0.000, C 0.000 }
gfCNCPoint5[13624] = {X 555.6452, Y 4.8909, Z -7.1667, A 0.000, B 0.000, C 0.000 }
gfCNCPoint5[13625] = {X 555.6478, Y 4.7819, Z -7.1667, A 0.000, B 0.000, C 0.000 }
gfCNCPoint5[13626] = {X 555.8079, Y 3.5173, Z -7.1667, A 0.000, B 0.000, C 0.000 }
gfCNCPoint5[13627] = {X 556.2012, Y 2.3049, Z -7.1667, A 0.000, B 0.000, C 0.000 }
gfCNCPoint5[13628] = {X 358.2606, Y 2.3049, Z -7.1667, A 0.000, B 0.000, C 0.000 }
gfCNCPoint5[13629] = {X 360.1223, Y 3.4745, Z -7.1667, A 0.000, B 0.000, C 0.000 }
gfCNCPoint5[13630] = {X 361.8553, Y 4.8275, Z -7.1667, A 0.000, B 0.000, C 0.000 }
gfCNCPoint5[13631] = {X 363.4418, Y 6.3497, Z -7.1667, A 0.000, B 0.000, C 0.000 }
gfCNCPoint5[13632] = {X 363.5020, Y 6.4140, Z -7.1667, A 0.000, B 0.000, C 0.000 }
gfCNCPoint5[13633] = {X 363.5619, Y 6.4784, Z -7.1667, A 0.000, B 0.000, C 0.000 }
gfCNCPoint5[13634] = {X 364.8933, Y 8.0616, Z -7.1667, A 0.000, B 0.000, C 0.000 }
gfCNCPoint5[13635] = {X 366.0915, Y 9.7477, Z -7.1667, A 0.000, B 0.000, C 0.000 }
gfCNCPoint5[13636] = {X 367.1486, Y 11.5257, Z -7.1667, A 0.000, B 0.000, C 0.000 }
gfCNCPoint5[13637] = {X 368.0576, Y 13.3838, Z -7.1667, A 0.000, B 0.000, C 0.000 }
gfCNCPoint5[13638] = {X 368.8125, Y 15.3097, Z -7.1667, A 0.000, B 0.000, C 0.000 }
gfCNCPoint5[13639] = {X 369.4082, Y 17.2905, Z -7.1667, A 0.000, B 0.000, C 0.000 }
gfCNCPoint5[13640] = {X 369.8993, Y 19.6245, Z -7.1667, A 0.000, B 0.000, C 0.000 }
gfCNCPoint5[13641] = {X 370.2160, Y 21.9884, Z -7.1667, A 0.000, B 0.000, C 0.000 }
gfCNCPoint5[13642] = {X 370.3566, Y 24.3693, Z -7.1667, A 0.000, B 0.000, C 0.000 }
gfCNCPoint5[13643] = {X 370.3203, Y 26.7540, Z -7.1667, A 0.000, B 0.000, C 0.000 }
gfCNCPoint5[13644] = {X 370.1073, Y 29.1295, Z -7.1667, A 0.000, B 0.000, C 0.000 }
gfCNCPoint5[13645] = {X 369.7188, Y 31.4827, Z -7.1667, A 0.000, B 0.000, C 0.000 }
gfCNCPoint5[13646] = {X 369.1829, Y 33.6343, Z -7.1667, A 0.000, B 0.000, C 0.000 }
gfCNCPoint5[13647] = {X 368.4592, Y 35.7303, Z -7.1667, A 0.000, B 0.000, C 0.000 }
gfCNCPoint5[13648] = {X 367.5532, Y 37.7541, Z -7.1667, A 0.000, B 0.000, C 0.000 }
gfCNCPoint5[13649] = {X 366.4722, Y 39.6901, Z -7.1667, A 0.000, B 0.000, C 0.000 }
gfCNCPoint5[13650] = {X 365.2245, Y 41.5231, Z -7.1667, A 0.000, B 0.000, C 0.000 }
gfCNCPoint5[13651] = {X 363.7791, Y 43.2834, Z -7.1667, A 0.000, B 0.000, C 0.000 }
gfCNCPoint5[13652] = {X 362.1635, Y 44.8888, Z -7.1667, A 0.000, B 0.000, C 0.000 }
gfCNCPoint5[13653] = {X 360.3941, Y 46.3231, Z -7.1667, A 0.000, B 0.000, C 0.000 }
gfCNCPoint5[13654] = {X 358.4891, Y 47.5715, Z -7.1667, A 0.000, B 0.000, C 0.000 }
gfCNCPoint5[13655] = {X 356.4678, Y 48.6213, Z -7.1667, A 0.000, B 0.000, C 0.000 }
gfCNCPoint5[13656] = {X 354.6708, Y 49.3152, Z -7.1667, A 0.000, B 0.000, C 0.000 }
gfCNCPoint5[13657] = {X 352.8231, Y 49.8601, Z -7.1667, A 0.000, B 0.000, C 0.000 }
gfCNCPoint5[13658] = {X 350.9372, Y 50.2525, Z -7.1667, A 0.000, B 0.000, C 0.000 }
gfCNCPoint5[13659] = {X 349.0255, Y 50.4896, Z -7.1667, A 0.000, B 0.000, C 0.000 }
gfCNCPoint5[13660] = {X 347.1008, Y 50.5699, Z -7.1667, A 0.000, B 0.000, C 0.000 }
gfCNCPoint5[13661] = {X 344.9874, Y 50.5337, Z -7.1667, A 0.000, B 0.000, C 0.000 }
gfCNCPoint5[13662] = {X 342.8851, Y 50.3145, Z -7.1667, A 0.000, B 0.000, C 0.000 }
gfCNCPoint5[13663] = {X 340.8096, Y 49.9139, Z -7.1667, A 0.000, B 0.000, C 0.000 }
gfCNCPoint5[13664] = {X 338.7767, Y 49.3350, Z -7.1667, A 0.000, B 0.000, C 0.000 }
gfCNCPoint5[13665] = {X 336.8016, Y 48.5821, Z -7.1667, A 0.000, B 0.000, C 0.000 }
gfCNCPoint5[13666] = {X 334.8992, Y 47.6608, Z -7.1667, A 0.000, B 0.000, C 0.000 }
gfCNCPoint5[13667] = {X 333.3420, Y 46.7039, Z -7.1667, A 0.000, B 0.000, C 0.000 }
gfCNCPoint5[13668] = {X 331.8608, Y 45.6333, Z -7.1667, A 0.000, B 0.000, C 0.000 }
gfCNCPoint5[13669] = {X 330.4638, Y 44.4550, Z -7.1667, A 0.000, B 0.000, C 0.000 }
gfCNCPoint5[13670] = {X 329.4665, Y 44.4078, Z -7.1667, A 0.000, B 0.000, C 0.000 }
gfCNCPoint5[13671] = {X 328.4997, Y 44.1587, Z -7.1667, A 0.000, B 0.000, C 0.000 }
gfCNCPoint5[13672] = {X 327.6038, Y 43.7181, Z -7.1667, A 0.000, B 0.000, C 0.000 }
gfCNCPoint5[13673] = {X 326.8164, Y 43.1044, Z -7.1667, A 0.000, B 0.000, C 0.000 }
gfCNCPoint5[13674] = {X 326.1897, Y 42.4934, Z -7.1667, A 0.000, B 0.000, C 0.000 }
gfCNCPoint5[13675] = {X 325.5686, Y 41.7541, Z -7.1667, A 0.000, B 0.000, C 0.000 }
gfCNCPoint5[13676] = {X 325.1052, Y 40.9070, Z -7.1667, A 0.000, B 0.000, C 0.000 }
gfCNCPoint5[13677] = {X 324.8177, Y 39.9852, Z -7.1667, A 0.000, B 0.000, C 0.000 }
gfCNCPoint5[13678] = {X 324.7172, Y 39.0249, Z -7.1667, A 0.000, B 0.000, C 0.000 }
gfCNCPoint5[13679] = {X 324.8079, Y 38.0635, Z -7.1667, A 0.000, B 0.000, C 0.000 }
gfCNCPoint5[13680] = {X 325.0860, Y 37.1389, Z -7.1667, A 0.000, B 0.000, C 0.000 }
gfCNCPoint5[13681] = {X 325.5408, Y 36.2871, Z -7.1667, A 0.000, B 0.000, C 0.000 }
gfCNCPoint5[13682] = {X 329.7765, Y 29.9537, Z -7.1667, A 0.000, B 0.000, C 0.000 }
gfCNCPoint5[13683] = {X 330.4614, Y 29.1399, Z -7.1667, A 0.000, B 0.000, C 0.000 }
gfCNCPoint5[13684] = {X 331.3063, Y 28.4938, Z -7.1667, A 0.000, B 0.000, C 0.000 }
gfCNCPoint5[13685] = {X 332.2712, Y 28.0462, Z -7.1667, A 0.000, B 0.000, C 0.000 }
gfCNCPoint5[13686] = {X 333.3101, Y 27.8182, Z -7.1667, A 0.000, B 0.000, C 0.000 }
gfCNCPoint5[13687] = {X 334.3737, Y 27.8207, Z -7.1667, A 0.000, B 0.000, C 0.000 }
gfCNCPoint5[13688] = {X 335.4115, Y 28.0536, Z -7.1667, A 0.000, B 0.000, C 0.000 }
gfCNCPoint5[13689] = {X 336.3743, Y 28.5058, Z -7.1667, A 0.000, B 0.000, C 0.000 }
gfCNCPoint5[13690] = {X 337.2161, Y 29.1559, Z -7.1667, A 0.000, B 0.000, C 0.000 }
gfCNCPoint5[13691] = {X 337.8208, Y 29.7387, Z -7.1667, A 0.000, B 0.000, C 0.000 }
gfCNCPoint5[13692] = {X 338.4966, Y 30.5667, Z -7.1667, A 0.000, B 0.000, C 0.000 }
gfCNCPoint5[13693] = {X 338.9759, Y 31.5220, Z -7.1667, A 0.000, B 0.000, C 0.000 }
gfCNCPoint5[13694] = {X 339.2358, Y 32.5587, Z -7.1667, A 0.000, B 0.000, C 0.000 }
gfCNCPoint5[13695] = {X 339.2638, Y 33.6271, Z -7.1667, A 0.000, B 0.000, C 0.000 }
gfCNCPoint5[13696] = {X 339.8712, Y 34.1824, Z -7.1667, A 0.000, B 0.000, C 0.000 }
gfCNCPoint5[13697] = {X 340.9506, Y 35.0427, Z -7.1667, A 0.000, B 0.000, C 0.000 }
gfCNCPoint5[13698] = {X 342.1369, Y 35.7481, Z -7.1667, A 0.000, B 0.000, C 0.000 }
gfCNCPoint5[13699] = {X 343.4081, Y 36.2857, Z -7.1667, A 0.000, B 0.000, C 0.000 }
gfCNCPoint5[13700] = {X 344.7407, Y 36.6454, Z -7.1667, A 0.000, B 0.000, C 0.000 }
gfCNCPoint5[13701] = {X 346.1097, Y 36.8205, Z -7.1667, A 0.000, B 0.000, C 0.000 }
gfCNCPoint5[13702] = {X 347.4899, Y 36.8078, Z -7.1667, A 0.000, B 0.000, C 0.000 }
gfCNCPoint5[13703] = {X 348.8395, Y 36.6266, Z -7.1667, A 0.000, B 0.000, C 0.000 }
gfCNCPoint5[13704] = {X 350.1415, Y 36.2280, Z -7.1667, A 0.000, B 0.000, C 0.000 }
gfCNCPoint5[13705] = {X 351.3612, Y 35.6228, Z -7.1667, A 0.000, B 0.000, C 0.000 }
gfCNCPoint5[13706] = {X 352.4661, Y 34.8269, Z -7.1667, A 0.000, B 0.000, C 0.000 }
gfCNCPoint5[13707] = {X 353.5668, Y 33.7573, Z -7.1667, A 0.000, B 0.000, C 0.000 }
gfCNCPoint5[13708] = {X 354.5194, Y 32.5540, Z -7.1667, A 0.000, B 0.000, C 0.000 }
gfCNCPoint5[13709] = {X 355.3078, Y 31.2371, Z -7.1667, A 0.000, B 0.000, C 0.000 }
gfCNCPoint5[13710] = {X 355.9186, Y 29.8291, Z -7.1667, A 0.000, B 0.000, C 0.000 }
gfCNCPoint5[13711] = {X 356.3416, Y 28.3538, Z -7.1667, A 0.000, B 0.000, C 0.000 }
gfCNCPoint5[13712] = {X 356.6061, Y 26.7186, Z -7.1667, A 0.000, B 0.000, C 0.000 }
gfCNCPoint5[13713] = {X 356.7138, Y 25.0657, Z -7.1667, A 0.000, B 0.000, C 0.000 }
gfCNCPoint5[13714] = {X 356.6637, Y 23.4100, Z -7.1667, A 0.000, B 0.000, C 0.000 }
gfCNCPoint5[13715] = {X 356.4563, Y 21.7666, Z -7.1667, A 0.000, B 0.000, C 0.000 }
gfCNCPoint5[13716] = {X 356.1196, Y 20.3211, Z -7.1667, A 0.000, B 0.000, C 0.000 }
gfCNCPoint5[13717] = {X 355.5960, Y 18.9323, Z -7.1667, A 0.000, B 0.000, C 0.000 }
gfCNCPoint5[13718] = {X 354.8946, Y 17.6242, Z -7.1667, A 0.000, B 0.000, C 0.000 }
gfCNCPoint5[13719] = {X 354.0274, Y 16.4197, Z -7.1667, A 0.000, B 0.000, C 0.000 }
gfCNCPoint5[13720] = {X 353.2099, Y 15.5488, Z -7.1667, A 0.000, B 0.000, C 0.000 }
gfCNCPoint5[13721] = {X 352.2795, Y 14.7997, Z -7.1667, A 0.000, B 0.000, C 0.000 }
gfCNCPoint5[13722] = {X 351.2542, Y 14.1869, Z -7.1667, A 0.000, B 0.000, C 0.000 }
gfCNCPoint5[13723] = {X 350.1538, Y 13.7223, Z -7.1667, A 0.000, B 0.000, C 0.000 }
gfCNCPoint5[13724] = {X 348.9995, Y 13.4149, Z -7.1667, A 0.000, B 0.000, C 0.000 }
gfCNCPoint5[13725] = {X 347.3622, Y 13.2071, Z -7.1667, A 0.000, B 0.000, C 0.000 }
gfCNCPoint5[13726] = {X 345.7117, Y 13.2118, Z -7.1667, A 0.000, B 0.000, C 0.000 }
gfCNCPoint5[13727] = {X 344.0755, Y 13.4287, Z -7.1667, A 0.000, B 0.000, C 0.000 }
gfCNCPoint5[13728] = {X 342.4808, Y 13.8544, Z -7.1667, A 0.000, B 0.000, C 0.000 }
gfCNCPoint5[13729] = {X 340.9542, Y 14.4817, Z -7.1667, A 0.000, B 0.000, C 0.000 }
gfCNCPoint5[13730] = {X 339.5209, Y 15.3002, Z -7.1667, A 0.000, B 0.000, C 0.000 }
gfCNCPoint5[13731] = {X 339.4271, Y 16.1858, Z -7.1667, A 0.000, B 0.000, C 0.000 }
gfCNCPoint5[13732] = {X 339.1738, Y 17.0396, Z -7.1667, A 0.000, B 0.000, C 0.000 }
gfCNCPoint5[13733] = {X 338.7697, Y 17.8331, Z -7.1667, A 0.000, B 0.000, C 0.000 }
gfCNCPoint5[13734] = {X 338.2280, Y 18.5399, Z -7.1667, A 0.000, B 0.000, C 0.000 }
gfCNCPoint5[13735] = {X 337.5670, Y 19.1366, Z -7.1667, A 0.000, B 0.000, C 0.000 }
gfCNCPoint5[13736] = {X 336.8399, Y 19.6716, Z -7.1667, A 0.000, B 0.000, C 0.000 }
gfCNCPoint5[13737] = {X 335.9170, Y 20.1909, Z -7.1667, A 0.000, B 0.000, C 0.000 }
gfCNCPoint5[13738] = {X 334.9039, Y 20.4988, Z -7.1667, A 0.000, B 0.000, C 0.000 }
gfCNCPoint5[13739] = {X 333.8481, Y 20.5809, Z -7.1667, A 0.000, B 0.000, C 0.000 }
gfCNCPoint5[13740] = {X 332.7995, Y 20.4334, Z -7.1667, A 0.000, B 0.000, C 0.000 }
gfCNCPoint5[13741] = {X 331.8074, Y 20.0631, Z -7.1667, A 0.000, B 0.000, C 0.000 }
gfCNCPoint5[13742] = {X 330.9186, Y 19.4875, Z -7.1667, A 0.000, B 0.000, C 0.000 }
gfCNCPoint5[13743] = {X 330.1748, Y 18.7338, Z -7.1667, A 0.000, B 0.000, C 0.000 }
gfCNCPoint5[13744] = {X 329.6111, Y 17.8373, Z -7.1667, A 0.000, B 0.000, C 0.000 }
gfCNCPoint5[13745] = {X 326.0906, Y 10.5950, Z -7.1667, A 0.000, B 0.000, C 0.000 }
gfCNCPoint5[13746] = {X 325.7555, Y 9.6856, Z -7.1667, A 0.000, B 0.000, C 0.000 }
gfCNCPoint5[13747] = {X 325.6067, Y 8.7279, Z -7.1667, A 0.000, B 0.000, C 0.000 }
gfCNCPoint5[13748] = {X 325.6502, Y 7.7596, Z -7.1667, A 0.000, B 0.000, C 0.000 }
gfCNCPoint5[13749] = {X 325.8842, Y 6.8191, Z -7.1667, A 0.000, B 0.000, C 0.000 }
gfCNCPoint5[13750] = {X 326.2994, Y 5.9433, Z -7.1667, A 0.000, B 0.000, C 0.000 }
gfCNCPoint5[13751] = {X 326.9295, Y 5.1131, Z -7.1667, A 0.000, B 0.000, C 0.000 }
gfCNCPoint5[13752] = {X 327.7216, Y 4.4356, Z -7.1667, A 0.000, B 0.000, C 0.000 }
gfCNCPoint5[13753] = {X 328.3967, Y 3.9733, Z -7.1667, A 0.000, B 0.000, C 0.000 }
gfCNCPoint5[13754] = {X 329.3291, Y 3.4829, Z -7.1667, A 0.000, B 0.000, C 0.000 }
gfCNCPoint5[13755] = {X 330.3450, Y 3.2041, Z -7.1667, A 0.000, B 0.000, C 0.000 }
gfCNCPoint5[13756] = {X 331.3970, Y 3.1498, Z -7.1667, A 0.000, B 0.000, C 0.000 }
gfCNCPoint5[13757] = {X 332.4362, Y 3.3225, Z -7.1667, A 0.000, B 0.000, C 0.000 }
gfCNCPoint5[13758] = {X 333.3719, Y 2.7963, Z -7.1667, A 0.000, B 0.000, C 0.000 }
gfCNCPoint5[13759] = {X 334.3265, Y 2.3049, Z -7.1667, A 0.000, B 0.000, C 0.000 }
gfCNCPoint5[13760] = {X 334.5383, Y 2.7356, Z -7.1667, A 0.000, B 0.000, C 0.000 }
gfCNCPoint5[13761] = {X 335.1906, Y 2.4250, Z -7.1667, A 0.000, B 0.000, C 0.000 }
gfCNCPoint5[13762] = {X 335.8506, Y 2.1310, Z -7.1667, A 0.000, B 0.000, C 0.000 }
gfCNCPoint5[13763] = {X 336.0151, Y 2.0600, Z -7.1667, A 0.000, B 0.000, C 0.000 }
gfCNCPoint5[13764] = {X 338.1041, Y 1.2614, Z -7.1667, A 0.000, B 0.000, C 0.000 }
gfCNCPoint5[13765] = {X 340.2533, Y 0.6425, Z -7.1667, A 0.000, B 0.000, C 0.000 }
gfCNCPoint5[13766] = {X 342.4471, Y 0.2078, Z -7.1667, A 0.000, B 0.000, C 0.000 }
gfCNCPoint5[13767] = {X 344.6698, Y -0.0397, Z -7.1667, A 0.000, B 0.000, C 0.000 }
gfCNCPoint5[13768] = {X 346.9055, Y -0.0982, Z -7.1667, A 0.000, B 0.000, C 0.000 }
gfCNCPoint5[13769] = {X 349.1382, Y 0.0328, Z -7.1667, A 0.000, B 0.000, C 0.000 }
gfCNCPoint5[13770] = {X 351.3517, Y 0.3523, Z -7.1667, A 0.000, B 0.000, C 0.000 }
gfCNCPoint5[13771] = {X 351.8890, Y 0.4533, Z -7.1667, A 0.000, B 0.000, C 0.000 }
gfCNCPoint5[13772] = {X 354.0188, Y 0.9989, Z -7.1667, A 0.000, B 0.000, C 0.000 }
gfCNCPoint5[13773] = {X 356.0803, Y 1.7631, Z -7.1667, A 0.000, B 0.000, C 0.000 }
gfCNCPoint5[13774] = {X 358.0510, Y 2.7377, Z -7.1667, A 0.000, B 0.000, C 0.000 }
gfCNCPoint5[13775] = {X 359.9097, Y 3.9119, Z -7.1667, A 0.000, B 0.000, C 0.000 }
gfCNCPoint5[13776] = {X 361.6362, Y 5.2732, Z -7.1667, A 0.000, B 0.000, C 0.000 }
gfCNCPoint5[13777] = {X 363.2117, Y 6.8067, Z -7.1667, A 0.000, B 0.000, C 0.000 }
gfCNCPoint5[13778] = {X 364.7628, Y 8.6829, Z -7.1667, A 0.000, B 0.000, C 0.000 }
gfCNCPoint5[13779] = {X 366.1236, Y 10.7014, Z -7.1667, A 0.000, B 0.000, C 0.000 }
gfCNCPoint5[13780] = {X 367.2811, Y 12.8430, Z -7.1667, A 0.000, B 0.000, C 0.000 }
gfCNCPoint5[13781] = {X 368.2242, Y 15.0872, Z -7.1667, A 0.000, B 0.000, C 0.000 }
gfCNCPoint5[13782] = {X 368.9440, Y 17.4127, Z -7.1667, A 0.000, B 0.000, C 0.000 }
gfCNCPoint5[13783] = {X 369.4272, Y 19.7109, Z -7.1667, A 0.000, B 0.000, C 0.000 }
gfCNCPoint5[13784] = {X 369.7387, Y 22.0385, Z -7.1667, A 0.000, B 0.000, C 0.000 }
gfCNCPoint5[13785] = {X 369.8768, Y 24.3829, Z -7.1667, A 0.000, B 0.000, C 0.000 }
gfCNCPoint5[13786] = {X 369.8409, Y 26.7310, Z -7.1667, A 0.000, B 0.000, C 0.000 }
gfCNCPoint5[13787] = {X 369.6310, Y 29.0700, Z -7.1667, A 0.000, B 0.000, C 0.000 }
gfCNCPoint5[13788] = {X 369.2484, Y 31.3870, Z -7.1667, A 0.000, B 0.000, C 0.000 }
gfCNCPoint5[13789] = {X 368.7226, Y 33.4980, Z -7.1667, A 0.000, B 0.000, C 0.000 }
gfCNCPoint5[13790] = {X 368.0125, Y 35.5544, Z -7.1667, A 0.000, B 0.000, C 0.000 }
gfCNCPoint5[13791] = {X 367.1236, Y 37.5400, Z -7.1667, A 0.000, B 0.000, C 0.000 }
gfCNCPoint5[13792] = {X 366.0628, Y 39.4394, Z -7.1667, A 0.000, B 0.000, C 0.000 }
gfCNCPoint5[13793] = {X 364.8385, Y 41.2377, Z -7.1667, A 0.000, B 0.000, C 0.000 }
gfCNCPoint5[13794] = {X 364.7204, Y 41.3991, Z -7.1667, A 0.000, B 0.000, C 0.000 }
gfCNCPoint5[13795] = {X 363.4201, Y 42.9679, Z -7.1667, A 0.000, B 0.000, C 0.000 }
gfCNCPoint5[13796] = {X 361.9805, Y 44.4100, Z -7.1667, A 0.000, B 0.000, C 0.000 }
gfCNCPoint5[13797] = {X 360.4141, Y 45.7132, Z -7.1667, A 0.000, B 0.000, C 0.000 }
gfCNCPoint5[13798] = {X 358.7341, Y 46.8663, Z -7.1667, A 0.000, B 0.000, C 0.000 }
gfCNCPoint5[13799] = {X 356.9549, Y 47.8595, Z -7.1667, A 0.000, B 0.000, C 0.000 }
gfCNCPoint5[13800] = {X 356.2499, Y 48.1931, Z -7.1667, A 0.000, B 0.000, C 0.000 }
gfCNCPoint5[13801] = {X 354.0456, Y 49.0155, Z -7.1667, A 0.000, B 0.000, C 0.000 }
gfCNCPoint5[13802] = {X 351.7691, Y 49.6095, Z -7.1667, A 0.000, B 0.000, C 0.000 }
gfCNCPoint5[13803] = {X 349.4440, Y 49.9689, Z -7.1667, A 0.000, B 0.000, C 0.000 }
gfCNCPoint5[13804] = {X 347.0943, Y 50.0899, Z -7.1667, A 0.000, B 0.000, C 0.000 }
gfCNCPoint5[13805] = {X 345.0202, Y 50.0548, Z -7.1667, A 0.000, B 0.000, C 0.000 }
gfCNCPoint5[13806] = {X 342.9569, Y 49.8399, Z -7.1667, A 0.000, B 0.000, C 0.000 }
gfCNCPoint5[13807] = {X 340.9200, Y 49.4467, Z -7.1667, A 0.000, B 0.000, C 0.000 }
gfCNCPoint5[13808] = {X 338.9249, Y 48.8784, Z -7.1667, A 0.000, B 0.000, C 0.000 }
gfCNCPoint5[13809] = {X 336.9867, Y 48.1391, Z -7.1667, A 0.000, B 0.000, C 0.000 }
gfCNCPoint5[13810] = {X 335.1199, Y 47.2344, Z -7.1667, A 0.000, B 0.000, C 0.000 }
gfCNCPoint5[13811] = {X 333.5417, Y 46.2601, Z -7.1667, A 0.000, B 0.000, C 0.000 }
gfCNCPoint5[13812] = {X 332.0436, Y 45.1665, Z -7.1667, A 0.000, B 0.000, C 0.000 }
gfCNCPoint5[13813] = {X 330.6346, Y 43.9603, Z -7.1667, A 0.000, B 0.000, C 0.000 }
gfCNCPoint5[13814] = {X 329.6761, Y 43.9518, Z -7.1667, A 0.000, B 0.000, C 0.000 }
gfCNCPoint5[13815] = {X 328.7421, Y 43.7359, Z -7.1667, A 0.000, B 0.000, C 0.000 }
gfCNCPoint5[13816] = {X 327.8770, Y 43.3228, Z -7.1667, A 0.000, B 0.000, C 0.000 }
gfCNCPoint5[13817] = {X 327.1220, Y 42.7322, Z -7.1667, A 0.000, B 0.000, C 0.000 }
gfCNCPoint5[13818] = {X 326.5249, Y 42.1498, Z -7.1667, A 0.000, B 0.000, C 0.000 }
gfCNCPoint5[13819] = {X 325.8848, Y 41.3619, Z -7.1667, A 0.000, B 0.000, C 0.000 }
gfCNCPoint5[13820] = {X 325.4424, Y 40.4483, Z -7.1667, A 0.000, B 0.000, C 0.000 }
gfCNCPoint5[13821] = {X 325.2210, Y 39.4576, Z -7.1667, A 0.000, B 0.000, C 0.000 }
gfCNCPoint5[13822] = {X 325.2326, Y 38.4426, Z -7.1667, A 0.000, B 0.000, C 0.000 }
gfCNCPoint5[13823] = {X 325.4765, Y 37.4572, Z -7.1667, A 0.000, B 0.000, C 0.000 }
gfCNCPoint5[13824] = {X 325.9397, Y 36.5539, Z -7.1667, A 0.000, B 0.000, C 0.000 }
gfCNCPoint5[13825] = {X 330.1988, Y 30.1861, Z -7.1667, A 0.000, B 0.000, C 0.000 }
gfCNCPoint5[13826] = {X 330.8195, Y 29.4619, Z -7.1667, A 0.000, B 0.000, C 0.000 }
gfCNCPoint5[13827] = {X 331.5816, Y 28.8884, Z -7.1667, A 0.000, B 0.000, C 0.000 }
gfCNCPoint5[13828] = {X 332.4494, Y 28.4927, Z -7.1667, A 0.000, B 0.000, C 0.000 }
gfCNCPoint5[13829] = {X 333.3822, Y 28.2932, Z -7.1667, A 0.000, B 0.000, C 0.000 }
gfCNCPoint5[13830] = {X 334.3359, Y 28.2995, Z -7.1667, A 0.000, B 0.000, C 0.000 }
gfCNCPoint5[13831] = {X 335.2660, Y 28.5111, Z -7.1667, A 0.000, B 0.000, C 0.000 }
gfCNCPoint5[13832] = {X 336.1285, Y 28.9182, Z -7.1667, A 0.000, B 0.000, C 0.000 }
gfCNCPoint5[13833] = {X 336.8831, Y 29.5016, Z -7.1667, A 0.000, B 0.000, C 0.000 }
gfCNCPoint5[13834] = {X 337.4845, Y 30.0811, Z -7.1667, A 0.000, B 0.000, C 0.000 }
gfCNCPoint5[13835] = {X 338.1249, Y 30.8765, Z -7.1667, A 0.000, B 0.000, C 0.000 }
gfCNCPoint5[13836] = {X 338.5648, Y 31.7980, Z -7.1667, A 0.000, B 0.000, C 0.000 }
gfCNCPoint5[13837] = {X 338.7804, Y 32.7961, Z -7.1667, A 0.000, B 0.000, C 0.000 }
gfCNCPoint5[13838] = {X 338.7601, Y 33.8170, Z -7.1667, A 0.000, B 0.000, C 0.000 }
gfCNCPoint5[13839] = {X 339.5473, Y 34.5367, Z -7.1667, A 0.000, B 0.000, C 0.000 }
gfCNCPoint5[13840] = {X 340.6403, Y 35.4108, Z -7.1667, A 0.000, B 0.000, C 0.000 }
gfCNCPoint5[13841] = {X 341.8388, Y 36.1334, Z -7.1667, A 0.000, B 0.000, C 0.000 }
gfCNCPoint5[13842] = {X 343.1220, Y 36.6919, Z -7.1667, A 0.000, B 0.000, C 0.000 }
gfCNCPoint5[13843] = {X 344.4676, Y 37.0766, Z -7.1667, A 0.000, B 0.000, C 0.000 }
gfCNCPoint5[13844] = {X 345.8522, Y 37.2808, Z -7.1667, A 0.000, B 0.000, C 0.000 }
gfCNCPoint5[13845] = {X 347.2516, Y 37.3008, Z -7.1667, A 0.000, B 0.000, C 0.000 }
gfCNCPoint5[13846] = {X 347.5147, Y 37.2872, Z -7.1667, A 0.000, B 0.000, C 0.000 }
gfCNCPoint5[13847] = {X 348.9420, Y 37.0955, Z -7.1667, A 0.000, B 0.000, C 0.000 }
gfCNCPoint5[13848] = {X 350.3190, Y 36.6740, Z -7.1667, A 0.000, B 0.000, C 0.000 }
gfCNCPoint5[13849] = {X 351.6090, Y 36.0339, Z -7.1667, A 0.000, B 0.000, C 0.000 }
gfCNCPoint5[13850] = {X 352.7776, Y 35.1922, Z -7.1667, A 0.000, B 0.000, C 0.000 }
gfCNCPoint5[13851] = {X 353.9232, Y 34.0789, Z -7.1667, A 0.000, B 0.000, C 0.000 }
gfCNCPoint5[13852] = {X 354.9147, Y 32.8263, Z -7.1667, A 0.000, B 0.000, C 0.000 }
gfCNCPoint5[13853] = {X 355.7352, Y 31.4556, Z -7.1667, A 0.000, B 0.000, C 0.000 }
gfCNCPoint5[13854] = {X 356.3709, Y 29.9900, Z -7.1667, A 0.000, B 0.000, C 0.000 }
gfCNCPoint5[13855] = {X 356.8109, Y 28.4543, Z -7.1667, A 0.000, B 0.000, C 0.000 }
gfCNCPoint5[13856] = {X 357.0830, Y 26.7727, Z -7.1667, A 0.000, B 0.000, C 0.000 }
gfCNCPoint5[13857] = {X 357.1937, Y 25.0729, Z -7.1667, A 0.000, B 0.000, C 0.000 }
gfCNCPoint5[13858] = {X 357.1420, Y 23.3702, Z -7.1667, A 0.000, B 0.000, C 0.000 }
gfCNCPoint5[13859] = {X 356.9284, Y 21.6801, Z -7.1667, A 0.000, B 0.000, C 0.000 }
gfCNCPoint5[13860] = {X 356.5768, Y 20.1749, Z -7.1667, A 0.000, B 0.000, C 0.000 }
gfCNCPoint5[13861] = {X 356.0308, Y 18.7288, Z -7.1667, A 0.000, B 0.000, C 0.000 }
gfCNCPoint5[13862] = {X 355.2998, Y 17.3669, Z -7.1667, A 0.000, B 0.000, C 0.000 }
gfCNCPoint5[13863] = {X 354.3964, Y 16.1126, Z -7.1667, A 0.000, B 0.000, C 0.000 }
gfCNCPoint5[13864] = {X 353.5334, Y 15.1941, Z -7.1667, A 0.000, B 0.000, C 0.000 }
gfCNCPoint5[13865] = {X 352.5515, Y 14.4042, Z -7.1667, A 0.000, B 0.000, C 0.000 }
gfCNCPoint5[13866] = {X 351.4695, Y 13.7579, Z -7.1667, A 0.000, B 0.000, C 0.000 }
gfCNCPoint5[13867] = {X 350.3084, Y 13.2679, Z -7.1667, A 0.000, B 0.000, C 0.000 }
gfCNCPoint5[13868] = {X 349.0905, Y 12.9436, Z -7.1667, A 0.000, B 0.000, C 0.000 }
gfCNCPoint5[13869] = {X 347.3478, Y 12.7254, Z -7.1667, A 0.000, B 0.000, C 0.000 }
gfCNCPoint5[13870] = {X 345.5916, Y 12.7391, Z -7.1667, A 0.000, B 0.000, C 0.000 }
gfCNCPoint5[13871] = {X 343.8525, Y 12.9844, Z -7.1667, A 0.000, B 0.000, C 0.000 }
gfCNCPoint5[13872] = {X 342.1610, Y 13.4570, Z -7.1667, A 0.000, B 0.000, C 0.000 }
gfCNCPoint5[13873] = {X 340.5466, Y 14.1486, Z -7.1667, A 0.000, B 0.000, C 0.000 }
gfCNCPoint5[13874] = {X 339.0376, Y 15.0473, Z -7.1667, A 0.000, B 0.000, C 0.000 }
gfCNCPoint5[13875] = {X 338.9895, Y 15.9050, Z -7.1667, A 0.000, B 0.000, C 0.000 }
gfCNCPoint5[13876] = {X 338.7756, Y 16.7370, Z -7.1667, A 0.000, B 0.000, C 0.000 }
gfCNCPoint5[13877] = {X 338.4041, Y 17.5116, Z -7.1667, A 0.000, B 0.000, C 0.000 }
gfCNCPoint5[13878] = {X 337.8892, Y 18.1993, Z -7.1667, A 0.000, B 0.000, C 0.000 }
gfCNCPoint5[13879] = {X 337.2504, Y 18.7738, Z -7.1667, A 0.000, B 0.000, C 0.000 }
gfCNCPoint5[13880] = {X 336.5606, Y 19.2813, Z -7.1667, A 0.000, B 0.000, C 0.000 }
gfCNCPoint5[13881] = {X 335.7284, Y 19.7495, Z -7.1667, A 0.000, B 0.000, C 0.000 }
gfCNCPoint5[13882] = {X 334.8148, Y 20.0271, Z -7.1667, A 0.000, B 0.000, C 0.000 }
gfCNCPoint5[13883] = {X 333.8628, Y 20.1012, Z -7.1667, A 0.000, B 0.000, C 0.000 }
gfCNCPoint5[13884] = {X 332.9173, Y 19.9681, Z -7.1667, A 0.000, B 0.000, C 0.000 }
gfCNCPoint5[13885] = {X 332.0228, Y 19.6341, Z -7.1667, A 0.000, B 0.000, C 0.000 }
gfCNCPoint5[13886] = {X 331.2213, Y 19.1151, Z -7.1667, A 0.000, B 0.000, C 0.000 }
gfCNCPoint5[13887] = {X 330.5507, Y 18.4353, Z -7.1667, A 0.000, B 0.000, C 0.000 }
gfCNCPoint5[13888] = {X 330.0425, Y 17.6269, Z -7.1667, A 0.000, B 0.000, C 0.000 }
gfCNCPoint5[13889] = {X 326.5223, Y 10.3852, Z -7.1667, A 0.000, B 0.000, C 0.000 }
gfCNCPoint5[13890] = {X 326.2154, Y 9.5469, Z -7.1667, A 0.000, B 0.000, C 0.000 }
gfCNCPoint5[13891] = {X 326.0841, Y 8.6639, Z -7.1667, A 0.000, B 0.000, C 0.000 }
gfCNCPoint5[13892] = {X 326.1338, Y 7.7725, Z -7.1667, A 0.000, B 0.000, C 0.000 }
gfCNCPoint5[13893] = {X 326.3623, Y 6.9096, Z -7.1667, A 0.000, B 0.000, C 0.000 }
gfCNCPoint5[13894] = {X 326.7603, Y 6.1105, Z -7.1667, A 0.000, B 0.000, C 0.000 }
gfCNCPoint5[13895] = {X 327.3114, Y 5.4082, Z -7.1667, A 0.000, B 0.000, C 0.000 }
gfCNCPoint5[13896] = {X 327.9929, Y 4.8316, Z -7.1667, A 0.000, B 0.000, C 0.000 }
gfCNCPoint5[13897] = {X 328.6647, Y 4.3715, Z -7.1667, A 0.000, B 0.000, C 0.000 }
gfCNCPoint5[13898] = {X 329.5521, Y 3.9112, Z -7.1667, A 0.000, B 0.000, C 0.000 }
gfCNCPoint5[13899] = {X 330.5205, Y 3.6632, Z -7.1667, A 0.000, B 0.000, C 0.000 }
gfCNCPoint5[13900] = {X 331.5199, Y 3.6401, Z -7.1667, A 0.000, B 0.000, C 0.000 }
gfCNCPoint5[13901] = {X 332.4988, Y 3.8432, Z -7.1667, A 0.000, B 0.000, C 0.000 }
gfCNCPoint5[13902] = {X 333.5073, Y 3.2687, Z -7.1667, A 0.000, B 0.000, C 0.000 }
gfCNCPoint5[13903] = {X 334.5383, Y 2.7356, Z -7.1667, A 0.000, B 0.000, C 0.000 }
gfCNCPoint5[13904] = {X 334.3265, Y 2.3049, Z -7.1667, A 0.000, B 0.000, C 0.000 }
gfCNCPoint5[13905] = {X 2.3033, Y 2.3049, Z -7.1667, A 0.000, B 0.000, C 0.000 }
gfCNCPoint5[13906] = {X 2.3033, Y 6.8597, Z -7.1667, A 0.000, B 0.000, C 0.000 }
gfCNCPoint5[13907] = {X 2.4162, Y 6.8823, Z -7.1667, A 0.000, B 0.000, C 0.000 }
gfCNCPoint5[13908] = {X 4.7217, Y 6.0043, Z -7.1667, A 0.000, B 0.000, C 0.000 }
gfCNCPoint5[13909] = {X 7.0993, Y 5.3464, Z -7.1667, A 0.000, B 0.000, C 0.000 }
gfCNCPoint5[13910] = {X 9.5281, Y 4.9143, Z -7.1667, A 0.000, B 0.000, C 0.000 }
gfCNCPoint5[13911] = {X 11.9868, Y 4.7118, Z -7.1667, A 0.000, B 0.000, C 0.000 }
gfCNCPoint5[13912] = {X 14.4536, Y 4.7408, Z -7.1667, A 0.000, B 0.000, C 0.000 }
gfCNCPoint5[13913] = {X 16.9068, Y 5.0009, Z -7.1667, A 0.000, B 0.000, C 0.000 }
gfCNCPoint5[13914] = {X 18.9214, Y 5.4154, Z -7.1667, A 0.000, B 0.000, C 0.000 }
gfCNCPoint5[13915] = {X 20.8824, Y 6.0354, Z -7.1667, A 0.000, B 0.000, C 0.000 }
gfCNCPoint5[13916] = {X 22.7691, Y 6.8542, Z -7.1667, A 0.000, B 0.000, C 0.000 }
gfCNCPoint5[13917] = {X 24.4895, Y 7.8178, Z -7.1667, A 0.000, B 0.000, C 0.000 }
gfCNCPoint5[13918] = {X 26.1061, Y 8.9468, Z -7.1667, A 0.000, B 0.000, C 0.000 }
gfCNCPoint5[13919] = {X 27.4004, Y 10.0772, Z -7.1667, A 0.000, B 0.000, C 0.000 }
gfCNCPoint5[13920] = {X 28.5615, Y 11.3441, Z -7.1667, A 0.000, B 0.000, C 0.000 }
gfCNCPoint5[13921] = {X 29.5751, Y 12.7318, Z -7.1667, A 0.000, B 0.000, C 0.000 }
gfCNCPoint5[13922] = {X 30.4286, Y 14.2233, Z -7.1667, A 0.000, B 0.000, C 0.000 }
gfCNCPoint5[13923] = {X 31.1116, Y 15.8002, Z -7.1667, A 0.000, B 0.000, C 0.000 }
gfCNCPoint5[13924] = {X 31.6712, Y 17.7359, Z -7.1667, A 0.000, B 0.000, C 0.000 }
gfCNCPoint5[13925] = {X 32.0044, Y 19.7231, Z -7.1667, A 0.000, B 0.000, C 0.000 }
gfCNCPoint5[13926] = {X 32.1067, Y 21.7355, Z -7.1667, A 0.000, B 0.000, C 0.000 }
gfCNCPoint5[13927] = {X 31.9768, Y 23.7462, Z -7.1667, A 0.000, B 0.000, C 0.000 }
gfCNCPoint5[13928] = {X 31.6165, Y 25.7287, Z -7.1667, A 0.000, B 0.000, C 0.000 }
gfCNCPoint5[13929] = {X 31.1974, Y 27.1578, Z -7.1667, A 0.000, B 0.000, C 0.000 }
gfCNCPoint5[13930] = {X 30.6307, Y 28.5350, Z -7.1667, A 0.000, B 0.000, C 0.000 }
gfCNCPoint5[13931] = {X 29.9226, Y 29.8451, Z -7.1667, A 0.000, B 0.000, C 0.000 }
gfCNCPoint5[13932] = {X 29.0810, Y 31.0738, Z -7.1667, A 0.000, B 0.000, C 0.000 }
gfCNCPoint5[13933] = {X 29.6386, Y 31.7920, Z -7.1667, A 0.000, B 0.000, C 0.000 }
gfCNCPoint5[13934] = {X 30.0954, Y 32.5783, Z -7.1667, A 0.000, B 0.000, C 0.000 }
gfCNCPoint5[13935] = {X 33.1423, Y 38.8726, Z -7.1667, A 0.000, B 0.000, C 0.000 }
gfCNCPoint5[13936] = {X 33.5391, Y 39.8957, Z -7.1667, A 0.000, B 0.000, C 0.000 }
gfCNCPoint5[13937] = {X 33.7662, Y 40.9694, Z -7.1667, A 0.000, B 0.000, C 0.000 }
gfCNCPoint5[13938] = {X 33.8177, Y 42.0656, Z -7.1667, A 0.000, B 0.000, C 0.000 }
gfCNCPoint5[13939] = {X 33.7164, Y 43.0266, Z -7.1667, A 0.000, B 0.000, C 0.000 }
gfCNCPoint5[13940] = {X 33.4799, Y 43.9636, Z -7.1667, A 0.000, B 0.000, C 0.000 }
gfCNCPoint5[13941] = {X 33.1103, Y 44.8630, Z -7.1667, A 0.000, B 0.000, C 0.000 }
gfCNCPoint5[13942] = {X 32.6161, Y 45.7005, Z -7.1667, A 0.000, B 0.000, C 0.000 }
gfCNCPoint5[13943] = {X 32.0075, Y 46.4590, Z -7.1667, A 0.000, B 0.000, C 0.000 }
gfCNCPoint5[13944] = {X 31.2970, Y 47.1229, Z -7.1667, A 0.000, B 0.000, C 0.000 }
gfCNCPoint5[13945] = {X 30.7614, Y 47.5560, Z -7.1667, A 0.000, B 0.000, C 0.000 }
gfCNCPoint5[13946] = {X 29.8557, Y 48.1750, Z -7.1667, A 0.000, B 0.000, C 0.000 }
gfCNCPoint5[13947] = {X 28.8624, Y 48.6405, Z -7.1667, A 0.000, B 0.000, C 0.000 }
gfCNCPoint5[13948] = {X 27.8071, Y 48.9406, Z -7.1667, A 0.000, B 0.000, C 0.000 }
gfCNCPoint5[13949] = {X 26.7174, Y 49.0673, Z -7.1667, A 0.000, B 0.000, C 0.000 }
gfCNCPoint5[13950] = {X 25.6215, Y 49.0174, Z -7.1667, A 0.000, B 0.000, C 0.000 }
gfCNCPoint5[13951] = {X 23.9295, Y 49.8570, Z -7.1667, A 0.000, B 0.000, C 0.000 }
gfCNCPoint5[13952] = {X 22.1904, Y 50.5943, Z -7.1667, A 0.000, B 0.000, C 0.000 }
gfCNCPoint5[13953] = {X 20.4105, Y 51.2267, Z -7.1667, A 0.000, B 0.000, C 0.000 }
gfCNCPoint5[13954] = {X 18.2617, Y 51.8322, Z -7.1667, A 0.000, B 0.000, C 0.000 }
gfCNCPoint5[13955] = {X 16.0678, Y 52.2454, Z -7.1667, A 0.000, B 0.000, C 0.000 }
gfCNCPoint5[13956] = {X 13.8460, Y 52.4631, Z -7.1667, A 0.000, B 0.000, C 0.000 }
gfCNCPoint5[13957] = {X 11.6137, Y 52.4837, Z -7.1667, A 0.000, B 0.000, C 0.000 }
gfCNCPoint5[13958] = {X 9.3882, Y 52.3068, Z -7.1667, A 0.000, B 0.000, C 0.000 }
gfCNCPoint5[13959] = {X 7.1871, Y 51.9340, Z -7.1667, A 0.000, B 0.000, C 0.000 }
gfCNCPoint5[13960] = {X 6.2987, Y 51.7237, Z -7.1667, A 0.000, B 0.000, C 0.000 }
gfCNCPoint5[13961] = {X 5.4213, Y 51.4713, Z -7.1667, A 0.000, B 0.000, C 0.000 }
gfCNCPoint5[13962] = {X 3.8340, Y 50.8959, Z -7.1667, A 0.000, B 0.000, C 0.000 }
gfCNCPoint5[13963] = {X 2.3033, Y 50.1832, Z -7.1667, A 0.000, B 0.000, C 0.000 }
gfCNCPoint5[13964] = {X 2.3033, Y 97.6951, Z -7.1667, A 0.000, B 0.000, C 0.000 }
gfCNCPoint5[13965] = {X 120.1200, Y 97.6951, Z -7.1667, A 0.000, B 0.000, C 0.000 }
gfCNCPoint5[13966] = {X 120.1200, Y 97.0659, Z -7.1667, A 0.000, B 0.000, C 0.000 }
gfCNCPoint5[13967] = {X 120.2337, Y 96.0187, Z -7.1667, A 0.000, B 0.000, C 0.000 }
gfCNCPoint5[13968] = {X 120.5695, Y 95.0202, Z -7.1667, A 0.000, B 0.000, C 0.000 }
gfCNCPoint5[13969] = {X 121.1117, Y 94.1171, Z -7.1667, A 0.000, B 0.000, C 0.000 }
gfCNCPoint5[13970] = {X 121.8351, Y 93.3514, Z -7.1667, A 0.000, B 0.000, C 0.000 }
gfCNCPoint5[13971] = {X 122.7060, Y 92.7587, Z -7.1667, A 0.000, B 0.000, C 0.000 }
gfCNCPoint5[13972] = {X 123.6838, Y 92.3668, Z -7.1667, A 0.000, B 0.000, C 0.000 }
gfCNCPoint5[13973] = {X 124.7228, Y 92.1938, Z -7.1667, A 0.000, B 0.000, C 0.000 }
gfCNCPoint5[13974] = {X 124.7837, Y 92.1780, Z -7.1667, A 0.000, B 0.000, C 0.000 }
gfCNCPoint5[13975] = {X 124.8455, Y 92.1665, Z -7.1667, A 0.000, B 0.000, C 0.000 }
gfCNCPoint5[13976] = {X 125.3649, Y 92.0895, Z -7.1667, A 0.000, B 0.000, C 0.000 }
gfCNCPoint5[13977] = {X 126.0999, Y 91.9684, Z -7.1667, A 0.000, B 0.000, C 0.000 }
gfCNCPoint5[13978] = {X 126.8256, Y 91.8009, Z -7.1667, A 0.000, B 0.000, C 0.000 }
gfCNCPoint5[13979] = {X 127.9390, Y 90.7470, Z -7.1667, A 0.000, B 0.000, C 0.000 }
gfCNCPoint5[13980] = {X 128.9957, Y 89.6363, Z -7.1667, A 0.000, B 0.000, C 0.000 }
gfCNCPoint5[13981] = {X 154.9457, Y 61.1414, Z -7.1667, A 0.000, B 0.000, C 0.000 }
gfCNCPoint5[13982] = {X 154.6591, Y 60.4490, Z -7.1667, A 0.000, B 0.000, C 0.000 }
gfCNCPoint5[13983] = {X 154.4818, Y 59.7210, Z -7.1667, A 0.000, B 0.000, C 0.000 }
gfCNCPoint5[13984] = {X 154.4181, Y 58.9744, Z -7.1667, A 0.000, B 0.000, C 0.000 }
gfCNCPoint5[13985] = {X 154.4180, Y 58.0000, Z -7.1667, A 0.000, B 0.000, C 0.000 }
gfCNCPoint5[13986] = {X 154.5117, Y 57.0480, Z -7.1667, A 0.000, B 0.000, C 0.000 }
gfCNCPoint5[13987] = {X 154.7894, Y 56.1325, Z -7.1667, A 0.000, B 0.000, C 0.000 }
gfCNCPoint5[13988] = {X 155.2404, Y 55.2888, Z -7.1667, A 0.000, B 0.000, C 0.000 }
gfCNCPoint5[13989] = {X 155.8473, Y 54.5493, Z -7.1667, A 0.000, B 0.000, C 0.000 }
gfCNCPoint5[13990] = {X 156.5868, Y 53.9424, Z -7.1667, A 0.000, B 0.000, C 0.000 }
gfCNCPoint5[13991] = {X 157.4305, Y 53.4915, Z -7.1667, A 0.000, B 0.000, C 0.000 }
gfCNCPoint5[13992] = {X 158.3459, Y 53.2138, Z -7.1667, A 0.000, B 0.000, C 0.000 }
gfCNCPoint5[13993] = {X 159.2980, Y 53.1200, Z -7.1667, A 0.000, B 0.000, C 0.000 }
gfCNCPoint5[13994] = {X 178.5335, Y 53.1200, Z -7.1667, A 0.000, B 0.000, C 0.000 }
gfCNCPoint5[13995] = {X 179.4855, Y 53.2138, Z -7.1667, A 0.000, B 0.000, C 0.000 }
gfCNCPoint5[13996] = {X 180.4010, Y 53.4915, Z -7.1667, A 0.000, B 0.000, C 0.000 }
gfCNCPoint5[13997] = {X 181.2447, Y 53.9424, Z -7.1667, A 0.000, B 0.000, C 0.000 }
gfCNCPoint5[13998] = {X 181.9842, Y 54.5493, Z -7.1667, A 0.000, B 0.000, C 0.000 }
gfCNCPoint5[13999] = {X 182.5911, Y 55.2888, Z -7.1667, A 0.000, B 0.000, C 0.000 }
gfCNCPoint5[14000] = {X 183.0420, Y 56.1325, Z -7.1667, A 0.000, B 0.000, C 0.000 }
gfCNCPoint5[14001] = {X 183.3197, Y 57.0480, Z -7.1667, A 0.000, B 0.000, C 0.000 }
gfCNCPoint5[14002] = {X 183.4135, Y 58.0000, Z -7.1667, A 0.000, B 0.000, C 0.000 }
gfCNCPoint5[14003] = {X 183.4133, Y 58.9744, Z -7.1667, A 0.000, B 0.000, C 0.000 }
gfCNCPoint5[14004] = {X 183.3513, Y 59.7110, Z -7.1667, A 0.000, B 0.000, C 0.000 }
gfCNCPoint5[14005] = {X 183.1786, Y 60.4298, Z -7.1667, A 0.000, B 0.000, C 0.000 }
gfCNCPoint5[14006] = {X 182.8994, Y 61.1142, Z -7.1667, A 0.000, B 0.000, C 0.000 }
gfCNCPoint5[14007] = {X 209.7093, Y 90.3814, Z -7.1667, A 0.000, B 0.000, C 0.000 }
gfCNCPoint5[14008] = {X 210.3600, Y 91.0553, Z -7.1667, A 0.000, B 0.000, C 0.000 }
gfCNCPoint5[14009] = {X 211.0451, Y 91.6941, Z -7.1667, A 0.000, B 0.000, C 0.000 }
gfCNCPoint5[14010] = {X 211.3188, Y 91.8793, Z -7.1667, A 0.000, B 0.000, C 0.000 }
gfCNCPoint5[14011] = {X 211.6306, Y 91.9884, Z -7.1667, A 0.000, B 0.000, C 0.000 }
gfCNCPoint5[14012] = {X 212.2004, Y 92.1083, Z -7.1667, A 0.000, B 0.000, C 0.000 }
gfCNCPoint5[14013] = {X 213.3849, Y 92.2575, Z -7.1667, A 0.000, B 0.000, C 0.000 }
gfCNCPoint5[14014] = {X 214.4294, Y 92.1757, Z -7.1667, A 0.000, B 0.000, C 0.000 }
gfCNCPoint5[14015] = {X 215.4754, Y 92.1154, Z -7.1667, A 0.000, B 0.000, C 0.000 }
gfCNCPoint5[14016] = {X 216.0504, Y 92.0562, Z -7.1667, A 0.000, B 0.000, C 0.000 }
gfCNCPoint5[14017] = {X 216.6043, Y 91.8909, Z -7.1667, A 0.000, B 0.000, C 0.000 }
gfCNCPoint5[14018] = {X 217.1177, Y 91.6253, Z -7.1667, A 0.000, B 0.000, C 0.000 }
gfCNCPoint5[14019] = {X 244.5999, Y 74.0197, Z -7.1667, A 0.000, B 0.000, C 0.000 }
gfCNCPoint5[14020] = {X 221.4279, Y 64.9268, Z -7.1667, A 0.000, B 0.000, C 0.000 }
gfCNCPoint5[14021] = {X 219.7198, Y 64.3546, Z -7.1667, A 0.000, B 0.000, C 0.000 }
gfCNCPoint5[14022] = {X 217.9576, Y 63.9811, Z -7.1667, A 0.000, B 0.000, C 0.000 }
gfCNCPoint5[14023] = {X 216.1643, Y 63.8112, Z -7.1667, A 0.000, B 0.000, C 0.000 }
gfCNCPoint5[14024] = {X 215.1118, Y 63.6594, Z -7.1667, A 0.000, B 0.000, C 0.000 }
gfCNCPoint5[14025] = {X 214.1172, Y 63.2831, Z -7.1667, A 0.000, B 0.000, C 0.000 }
gfCNCPoint5[14026] = {X 213.2277, Y 62.7004, Z -7.1667, A 0.000, B 0.000, C 0.000 }
gfCNCPoint5[14027] = {X 212.4855, Y 61.9388, Z -7.1667, A 0.000, B 0.000, C 0.000 }
gfCNCPoint5[14028] = {X 211.9260, Y 61.0345, Z -7.1667, A 0.000, B 0.000, C 0.000 }
gfCNCPoint5[14029] = {X 211.5756, Y 60.0305, Z -7.1667, A 0.000, B 0.000, C 0.000 }
gfCNCPoint5[14030] = {X 211.4510, Y 58.9744, Z -7.1667, A 0.000, B 0.000, C 0.000 }
gfCNCPoint5[14031] = {X 211.4508, Y 58.0000, Z -7.1667, A 0.000, B 0.000, C 0.000 }
gfCNCPoint5[14032] = {X 211.5446, Y 57.0480, Z -7.1667, A 0.000, B 0.000, C 0.000 }
gfCNCPoint5[14033] = {X 211.8223, Y 56.1325, Z -7.1667, A 0.000, B 0.000, C 0.000 }
gfCNCPoint5[14034] = {X 212.2732, Y 55.2888, Z -7.1667, A 0.000, B 0.000, C 0.000 }
gfCNCPoint5[14035] = {X 212.8801, Y 54.5493, Z -7.1667, A 0.000, B 0.000, C 0.000 }
gfCNCPoint5[14036] = {X 213.6196, Y 53.9424, Z -7.1667, A 0.000, B 0.000, C 0.000 }
gfCNCPoint5[14037] = {X 214.4633, Y 53.4915, Z -7.1667, A 0.000, B 0.000, C 0.000 }
gfCNCPoint5[14038] = {X 215.3788, Y 53.2138, Z -7.1667, A 0.000, B 0.000, C 0.000 }
gfCNCPoint5[14039] = {X 216.3308, Y 53.1200, Z -7.1667, A 0.000, B 0.000, C 0.000 }
gfCNCPoint5[14040] = {X 237.2617, Y 53.1200, Z -7.1667, A 0.000, B 0.000, C 0.000 }
gfCNCPoint5[14041] = {X 238.3264, Y 53.2376, Z -7.1667, A 0.000, B 0.000, C 0.000 }
gfCNCPoint5[14042] = {X 239.3399, Y 53.5846, Z -7.1667, A 0.000, B 0.000, C 0.000 }
gfCNCPoint5[14043] = {X 240.2532, Y 54.1444, Z -7.1667, A 0.000, B 0.000, C 0.000 }
gfCNCPoint5[14044] = {X 241.0223, Y 54.8900, Z -7.1667, A 0.000, B 0.000, C 0.000 }
gfCNCPoint5[14045] = {X 241.6103, Y 55.7854, Z -7.1667, A 0.000, B 0.000, C 0.000 }
gfCNCPoint5[14046] = {X 241.9887, Y 56.7876, Z -7.1667, A 0.000, B 0.000, C 0.000 }
gfCNCPoint5[14047] = {X 242.1393, Y 57.8481, Z -7.1667, A 0.000, B 0.000, C 0.000 }
gfCNCPoint5[14048] = {X 248.3224, Y 60.2592, Z -7.1667, A 0.000, B 0.000, C 0.000 }
gfCNCPoint5[14049] = {X 275.0718, Y 70.8765, Z -7.1667, A 0.000, B 0.000, C 0.000 }
gfCNCPoint5[14050] = {X 275.0716, Y 63.6739, Z -7.1667, A 0.000, B 0.000, C 0.000 }
gfCNCPoint5[14051] = {X 274.0635, Y 63.3055, Z -7.1667, A 0.000, B 0.000, C 0.000 }
gfCNCPoint5[14052] = {X 273.1604, Y 62.7255, Z -7.1667, A 0.000, B 0.000, C 0.000 }
gfCNCPoint5[14053] = {X 272.4058, Y 61.9622, Z -7.1667, A 0.000, B 0.000, C 0.000 }
gfCNCPoint5[14054] = {X 271.8364, Y 61.0524, Z -7.1667, A 0.000, B 0.000, C 0.000 }
gfCNCPoint5[14055] = {X 271.4797, Y 60.0401, Z -7.1667, A 0.000, B 0.000, C 0.000 }
gfCNCPoint5[14056] = {X 271.3529, Y 58.9744, Z -7.1667, A 0.000, B 0.000, C 0.000 }
gfCNCPoint5[14057] = {X 271.3527, Y 58.0000, Z -7.1667, A 0.000, B 0.000, C 0.000 }
gfCNCPoint5[14058] = {X 271.4465, Y 57.0480, Z -7.1667, A 0.000, B 0.000, C 0.000 }
gfCNCPoint5[14059] = {X 271.7242, Y 56.1325, Z -7.1667, A 0.000, B 0.000, C 0.000 }
gfCNCPoint5[14060] = {X 272.1751, Y 55.2888, Z -7.1667, A 0.000, B 0.000, C 0.000 }
gfCNCPoint5[14061] = {X 272.7820, Y 54.5493, Z -7.1667, A 0.000, B 0.000, C 0.000 }
gfCNCPoint5[14062] = {X 273.5215, Y 53.9424, Z -7.1667, A 0.000, B 0.000, C 0.000 }
gfCNCPoint5[14063] = {X 274.3652, Y 53.4915, Z -7.1667, A 0.000, B 0.000, C 0.000 }
gfCNCPoint5[14064] = {X 275.2806, Y 53.2138, Z -7.1667, A 0.000, B 0.000, C 0.000 }
gfCNCPoint5[14065] = {X 276.2327, Y 53.1200, Z -7.1667, A 0.000, B 0.000, C 0.000 }
gfCNCPoint5[14066] = {X 292.7731, Y 53.1200, Z -7.1667, A 0.000, B 0.000, C 0.000 }
gfCNCPoint5[14067] = {X 293.7251, Y 53.2138, Z -7.1667, A 0.000, B 0.000, C 0.000 }
gfCNCPoint5[14068] = {X 294.6406, Y 53.4915, Z -7.1667, A 0.000, B 0.000, C 0.000 }
gfCNCPoint5[14069] = {X 295.4843, Y 53.9424, Z -7.1667, A 0.000, B 0.000, C 0.000 }
gfCNCPoint5[14070] = {X 296.2238, Y 54.5493, Z -7.1667, A 0.000, B 0.000, C 0.000 }
gfCNCPoint5[14071] = {X 296.8307, Y 55.2888, Z -7.1667, A 0.000, B 0.000, C 0.000 }
gfCNCPoint5[14072] = {X 297.2816, Y 56.1325, Z -7.1667, A 0.000, B 0.000, C 0.000 }
gfCNCPoint5[14073] = {X 297.5593, Y 57.0480, Z -7.1667, A 0.000, B 0.000, C 0.000 }
gfCNCPoint5[14074] = {X 297.6531, Y 58.0000, Z -7.1667, A 0.000, B 0.000, C 0.000 }
gfCNCPoint5[14075] = {X 297.6531, Y 58.9365, Z -7.1667, A 0.000, B 0.000, C 0.000 }
gfCNCPoint5[14076] = {X 297.5312, Y 60.0089, Z -7.1667, A 0.000, B 0.000, C 0.000 }
gfCNCPoint5[14077] = {X 297.1773, Y 61.0285, Z -7.1667, A 0.000, B 0.000, C 0.000 }
gfCNCPoint5[14078] = {X 296.6086, Y 61.9458, Z -7.1667, A 0.000, B 0.000, C 0.000 }
gfCNCPoint5[14079] = {X 295.8527, Y 62.7162, Z -7.1667, A 0.000, B 0.000, C 0.000 }
gfCNCPoint5[14080] = {X 294.9464, Y 63.3023, Z -7.1667, A 0.000, B 0.000, C 0.000 }
gfCNCPoint5[14081] = {X 293.9338, Y 63.6755, Z -7.1667, A 0.000, B 0.000, C 0.000 }
gfCNCPoint5[14082] = {X 293.9338, Y 92.3193, Z -7.1667, A 0.000, B 0.000, C 0.000 }
gfCNCPoint5[14083] = {X 294.9456, Y 92.6948, Z -7.1667, A 0.000, B 0.000, C 0.000 }
gfCNCPoint5[14084] = {X 295.8510, Y 93.2823, Z -7.1667, A 0.000, B 0.000, C 0.000 }
gfCNCPoint5[14085] = {X 296.6062, Y 94.0532, Z -7.1667, A 0.000, B 0.000, C 0.000 }
gfCNCPoint5[14086] = {X 297.1749, Y 94.9705, Z -7.1667, A 0.000, B 0.000, C 0.000 }
gfCNCPoint5[14087] = {X 297.5296, Y 95.9898, Z -7.1667, A 0.000, B 0.000, C 0.000 }
gfCNCPoint5[14088] = {X 297.6531, Y 97.0620, Z -7.1667, A 0.000, B 0.000, C 0.000 }
gfCNCPoint5[14089] = {X 297.6531, Y 97.6951, Z -7.1667, A 0.000, B 0.000, C 0.000 }
gfCNCPoint5[14090] = {X 297.1731, Y 97.6951, Z -7.1667, A 0.000, B 0.000, C 0.000 }
gfCNCPoint5[14091] = {X 297.1731, Y 98.0000, Z -7.1667, A 0.000, B 0.000, C 0.000 }
gfCNCPoint5[14092] = {X 297.0628, Y 98.9791, Z -7.1667, A 0.000, B 0.000, C 0.000 }
gfCNCPoint5[14093] = {X 296.7373, Y 99.9091, Z -7.1667, A 0.000, B 0.000, C 0.000 }
gfCNCPoint5[14094] = {X 296.2131, Y 100.7434, Z -7.1667, A 0.000, B 0.000, C 0.000 }
gfCNCPoint5[14095] = {X 295.5164, Y 101.4401, Z -7.1667, A 0.000, B 0.000, C 0.000 }
gfCNCPoint5[14096] = {X 294.6822, Y 101.9643, Z -7.1667, A 0.000, B 0.000, C 0.000 }
gfCNCPoint5[14097] = {X 293.7522, Y 102.2897, Z -7.1667, A 0.000, B 0.000, C 0.000 }
gfCNCPoint5[14098] = {X 292.7731, Y 102.4000, Z -7.1667, A 0.000, B 0.000, C 0.000 }
gfCNCPoint5[14099] = {X 276.2327, Y 102.4000, Z -7.1667, A 0.000, B 0.000, C 0.000 }
gfCNCPoint5[14100] = {X 275.2536, Y 102.2897, Z -7.1667, A 0.000, B 0.000, C 0.000 }
gfCNCPoint5[14101] = {X 274.3236, Y 101.9643, Z -7.1667, A 0.000, B 0.000, C 0.000 }
gfCNCPoint5[14102] = {X 273.4893, Y 101.4401, Z -7.1667, A 0.000, B 0.000, C 0.000 }
gfCNCPoint5[14103] = {X 272.7926, Y 100.7434, Z -7.1667, A 0.000, B 0.000, C 0.000 }
gfCNCPoint5[14104] = {X 272.2684, Y 99.9091, Z -7.1667, A 0.000, B 0.000, C 0.000 }
gfCNCPoint5[14105] = {X 271.9430, Y 98.9791, Z -7.1667, A 0.000, B 0.000, C 0.000 }
gfCNCPoint5[14106] = {X 271.8327, Y 98.0000, Z -7.1667, A 0.000, B 0.000, C 0.000 }
gfCNCPoint5[14107] = {X 271.8329, Y 97.0190, Z -7.1667, A 0.000, B 0.000, C 0.000 }
gfCNCPoint5[14108] = {X 271.9305, Y 96.1432, Z -7.1667, A 0.000, B 0.000, C 0.000 }
gfCNCPoint5[14109] = {X 272.2006, Y 95.3045, Z -7.1667, A 0.000, B 0.000, C 0.000 }
gfCNCPoint5[14110] = {X 272.6325, Y 94.5364, Z -7.1667, A 0.000, B 0.000, C 0.000 }
gfCNCPoint5[14111] = {X 273.2087, Y 93.8698, Z -7.1667, A 0.000, B 0.000, C 0.000 }
gfCNCPoint5[14112] = {X 273.9062, Y 93.3313, Z -7.1667, A 0.000, B 0.000, C 0.000 }
gfCNCPoint5[14113] = {X 274.6970, Y 92.9426, Z -7.1667, A 0.000, B 0.000, C 0.000 }
gfCNCPoint5[14114] = {X 275.5494, Y 92.7193, Z -7.1667, A 0.000, B 0.000, C 0.000 }
gfCNCPoint5[14115] = {X 275.5494, Y 85.6495, Z -7.1667, A 0.000, B 0.000, C 0.000 }
gfCNCPoint5[14116] = {X 262.6483, Y 80.5923, Z -7.1667, A 0.000, B 0.000, C 0.000 }
gfCNCPoint5[14117] = {X 262.3213, Y 80.7989, Z -7.1667, A 0.000, B 0.000, C 0.000 }
gfCNCPoint5[14118] = {X 237.8776, Y 96.6317, Z -7.1667, A 0.000, B 0.000, C 0.000 }
gfCNCPoint5[14119] = {X 237.8798, Y 97.0659, Z -7.1667, A 0.000, B 0.000, C 0.000 }
gfCNCPoint5[14120] = {X 237.8798, Y 98.0000, Z -7.1667, A 0.000, B 0.000, C 0.000 }
gfCNCPoint5[14121] = {X 237.7695, Y 98.9791, Z -7.1667, A 0.000, B 0.000, C 0.000 }
gfCNCPoint5[14122] = {X 237.4440, Y 99.9091, Z -7.1667, A 0.000, B 0.000, C 0.000 }
gfCNCPoint5[14123] = {X 236.9198, Y 100.7434, Z -7.1667, A 0.000, B 0.000, C 0.000 }
gfCNCPoint5[14124] = {X 236.2231, Y 101.4401, Z -7.1667, A 0.000, B 0.000, C 0.000 }
gfCNCPoint5[14125] = {X 235.3889, Y 101.9643, Z -7.1667, A 0.000, B 0.000, C 0.000 }
gfCNCPoint5[14126] = {X 234.4589, Y 102.2897, Z -7.1667, A 0.000, B 0.000, C 0.000 }
gfCNCPoint5[14127] = {X 233.4798, Y 102.4000, Z -7.1667, A 0.000, B 0.000, C 0.000 }
gfCNCPoint5[14128] = {X 214.1790, Y 102.4000, Z -7.1667, A 0.000, B 0.000, C 0.000 }
gfCNCPoint5[14129] = {X 213.7862, Y 102.3824, Z -7.1667, A 0.000, B 0.000, C 0.000 }
gfCNCPoint5[14130] = {X 213.3966, Y 102.3299, Z -7.1667, A 0.000, B 0.000, C 0.000 }
gfCNCPoint5[14131] = {X 213.0069, Y 102.3824, Z -7.1667, A 0.000, B 0.000, C 0.000 }
gfCNCPoint5[14132] = {X 212.6141, Y 102.4000, Z -7.1667, A 0.000, B 0.000, C 0.000 }
gfCNCPoint5[14133] = {X 194.9870, Y 102.4000, Z -7.1667, A 0.000, B 0.000, C 0.000 }
gfCNCPoint5[14134] = {X 194.0079, Y 102.2897, Z -7.1667, A 0.000, B 0.000, C 0.000 }
gfCNCPoint5[14135] = {X 193.0779, Y 101.9643, Z -7.1667, A 0.000, B 0.000, C 0.000 }
gfCNCPoint5[14136] = {X 192.2436, Y 101.4401, Z -7.1667, A 0.000, B 0.000, C 0.000 }
gfCNCPoint5[14137] = {X 191.5469, Y 100.7434, Z -7.1667, A 0.000, B 0.000, C 0.000 }
gfCNCPoint5[14138] = {X 191.0227, Y 99.9091, Z -7.1667, A 0.000, B 0.000, C 0.000 }
gfCNCPoint5[14139] = {X 190.6973, Y 98.9791, Z -7.1667, A 0.000, B 0.000, C 0.000 }
gfCNCPoint5[14140] = {X 190.5870, Y 98.0000, Z -7.1667, A 0.000, B 0.000, C 0.000 }
gfCNCPoint5[14141] = {X 190.5870, Y 97.0659, Z -7.1667, A 0.000, B 0.000, C 0.000 }
gfCNCPoint5[14142] = {X 190.6897, Y 96.1207, Z -7.1667, A 0.000, B 0.000, C 0.000 }
gfCNCPoint5[14143] = {X 190.9931, Y 95.2196, Z -7.1667, A 0.000, B 0.000, C 0.000 }
gfCNCPoint5[14144] = {X 191.4830, Y 94.4047, Z -7.1667, A 0.000, B 0.000, C 0.000 }
gfCNCPoint5[14145] = {X 188.5295, Y 91.1802, Z -7.1667, A 0.000, B 0.000, C 0.000 }
gfCNCPoint5[14146] = {X 150.1254, Y 91.1802, Z -7.1667, A 0.000, B 0.000, C 0.000 }
gfCNCPoint5[14147] = {X 147.2503, Y 94.3655, Z -7.1667, A 0.000, B 0.000, C 0.000 }
gfCNCPoint5[14148] = {X 147.7564, Y 95.1896, Z -7.1667, A 0.000, B 0.000, C 0.000 }
gfCNCPoint5[14149] = {X 148.0711, Y 96.1041, Z -7.1667, A 0.000, B 0.000, C 0.000 }
gfCNCPoint5[14150] = {X 148.1791, Y 97.0652, Z -7.1667, A 0.000, B 0.000, C 0.000 }
gfCNCPoint5[14151] = {X 148.1791, Y 98.0000, Z -7.1667, A 0.000, B 0.000, C 0.000 }
gfCNCPoint5[14152] = {X 148.0688, Y 98.9791, Z -7.1667, A 0.000, B 0.000, C 0.000 }
gfCNCPoint5[14153] = {X 147.7434, Y 99.9091, Z -7.1667, A 0.000, B 0.000, C 0.000 }
gfCNCPoint5[14154] = {X 147.2192, Y 100.7434, Z -7.1667, A 0.000, B 0.000, C 0.000 }
gfCNCPoint5[14155] = {X 146.5225, Y 101.4401, Z -7.1667, A 0.000, B 0.000, C 0.000 }
gfCNCPoint5[14156] = {X 145.6882, Y 101.9643, Z -7.1667, A 0.000, B 0.000, C 0.000 }
gfCNCPoint5[14157] = {X 144.7582, Y 102.2897, Z -7.1667, A 0.000, B 0.000, C 0.000 }
gfCNCPoint5[14158] = {X 143.7791, Y 102.4000, Z -7.1667, A 0.000, B 0.000, C 0.000 }
gfCNCPoint5[14159] = {X 125.0000, Y 102.4000, Z -7.1667, A 0.000, B 0.000, C 0.000 }
gfCNCPoint5[14160] = {X 124.0209, Y 102.2897, Z -7.1667, A 0.000, B 0.000, C 0.000 }
gfCNCPoint5[14161] = {X 123.0909, Y 101.9643, Z -7.1667, A 0.000, B 0.000, C 0.000 }
gfCNCPoint5[14162] = {X 122.2566, Y 101.4401, Z -7.1667, A 0.000, B 0.000, C 0.000 }
gfCNCPoint5[14163] = {X 121.5599, Y 100.7434, Z -7.1667, A 0.000, B 0.000, C 0.000 }
gfCNCPoint5[14164] = {X 121.0357, Y 99.9091, Z -7.1667, A 0.000, B 0.000, C 0.000 }
gfCNCPoint5[14165] = {X 120.7103, Y 98.9791, Z -7.1667, A 0.000, B 0.000, C 0.000 }
gfCNCPoint5[14166] = {X 120.6000, Y 98.0000, Z -7.1667, A 0.000, B 0.000, C 0.000 }
gfCNCPoint5[14167] = {X 120.6000, Y 97.0659, Z -7.1667, A 0.000, B 0.000, C 0.000 }
gfCNCPoint5[14168] = {X 120.7045, Y 96.1125, Z -7.1667, A 0.000, B 0.000, C 0.000 }
gfCNCPoint5[14169] = {X 121.0132, Y 95.2043, Z -7.1667, A 0.000, B 0.000, C 0.000 }
gfCNCPoint5[14170] = {X 121.5113, Y 94.3847, Z -7.1667, A 0.000, B 0.000, C 0.000 }
gfCNCPoint5[14171] = {X 122.1753, Y 93.6924, Z -7.1667, A 0.000, B 0.000, C 0.000 }
gfCNCPoint5[14172] = {X 122.9734, Y 93.1604, Z -7.1667, A 0.000, B 0.000, C 0.000 }
gfCNCPoint5[14173] = {X 123.8679, Y 92.8141, Z -7.1667, A 0.000, B 0.000, C 0.000 }
gfCNCPoint5[14174] = {X 124.8161, Y 92.6698, Z -7.1667, A 0.000, B 0.000, C 0.000 }
gfCNCPoint5[14175] = {X 124.8651, Y 92.6523, Z -7.1667, A 0.000, B 0.000, C 0.000 }
gfCNCPoint5[14176] = {X 124.9160, Y 92.6413, Z -7.1667, A 0.000, B 0.000, C 0.000 }
gfCNCPoint5[14177] = {X 125.4412, Y 92.5635, Z -7.1667, A 0.000, B 0.000, C 0.000 }
gfCNCPoint5[14178] = {X 126.2565, Y 92.4265, Z -7.1667, A 0.000, B 0.000, C 0.000 }
gfCNCPoint5[14179] = {X 127.0607, Y 92.2347, Z -7.1667, A 0.000, B 0.000, C 0.000 }
gfCNCPoint5[14180] = {X 128.2379, Y 91.1268, Z -7.1667, A 0.000, B 0.000, C 0.000 }
gfCNCPoint5[14181] = {X 129.3532, Y 89.9565, Z -7.1667, A 0.000, B 0.000, C 0.000 }
gfCNCPoint5[14182] = {X 155.5323, Y 61.2101, Z -7.1667, A 0.000, B 0.000, C 0.000 }
gfCNCPoint5[14183] = {X 155.1838, Y 60.4941, Z -7.1667, A 0.000, B 0.000, C 0.000 }
gfCNCPoint5[14184] = {X 154.9700, Y 59.7271, Z -7.1667, A 0.000, B 0.000, C 0.000 }
gfCNCPoint5[14185] = {X 154.8980, Y 58.9341, Z -7.1667, A 0.000, B 0.000, C 0.000 }
gfCNCPoint5[14186] = {X 154.8980, Y 58.0000, Z -7.1667, A 0.000, B 0.000, C 0.000 }
gfCNCPoint5[14187] = {X 155.0083, Y 57.0209, Z -7.1667, A 0.000, B 0.000, C 0.000 }
gfCNCPoint5[14188] = {X 155.3337, Y 56.0909, Z -7.1667, A 0.000, B 0.000, C 0.000 }
gfCNCPoint5[14189] = {X 155.8579, Y 55.2566, Z -7.1667, A 0.000, B 0.000, C 0.000 }
gfCNCPoint5[14190] = {X 156.5546, Y 54.5599, Z -7.1667, A 0.000, B 0.000, C 0.000 }
gfCNCPoint5[14191] = {X 157.3889, Y 54.0357, Z -7.1667, A 0.000, B 0.000, C 0.000 }
gfCNCPoint5[14192] = {X 158.3189, Y 53.7103, Z -7.1667, A 0.000, B 0.000, C 0.000 }
gfCNCPoint5[14193] = {X 159.2980, Y 53.6000, Z -7.1667, A 0.000, B 0.000, C 0.000 }
gfCNCPoint5[14194] = {X 178.5335, Y 53.6000, Z -7.1667, A 0.000, B 0.000, C 0.000 }
gfCNCPoint5[14195] = {X 179.5126, Y 53.7103, Z -7.1667, A 0.000, B 0.000, C 0.000 }
gfCNCPoint5[14196] = {X 180.4426, Y 54.0357, Z -7.1667, A 0.000, B 0.000, C 0.000 }
gfCNCPoint5[14197] = {X 181.2769, Y 54.5599, Z -7.1667, A 0.000, B 0.000, C 0.000 }
gfCNCPoint5[14198] = {X 181.9736, Y 55.2566, Z -7.1667, A 0.000, B 0.000, C 0.000 }
gfCNCPoint5[14199] = {X 182.4978, Y 56.0909, Z -7.1667, A 0.000, B 0.000, C 0.000 }
gfCNCPoint5[14200] = {X 182.8232, Y 57.0209, Z -7.1667, A 0.000, B 0.000, C 0.000 }
gfCNCPoint5[14201] = {X 182.9335, Y 58.0000, Z -7.1667, A 0.000, B 0.000, C 0.000 }
gfCNCPoint5[14202] = {X 182.9334, Y 58.9704, Z -7.1667, A 0.000, B 0.000, C 0.000 }
gfCNCPoint5[14203] = {X 182.8588, Y 59.7415, Z -7.1667, A 0.000, B 0.000, C 0.000 }
gfCNCPoint5[14204] = {X 182.6501, Y 60.4876, Z -7.1667, A 0.000, B 0.000, C 0.000 }
gfCNCPoint5[14205] = {X 182.3138, Y 61.1856, Z -7.1667, A 0.000, B 0.000, C 0.000 }
gfCNCPoint5[14206] = {X 209.3554, Y 90.7056, Z -7.1667, A 0.000, B 0.000, C 0.000 }
gfCNCPoint5[14207] = {X 210.0236, Y 91.3976, Z -7.1667, A 0.000, B 0.000, C 0.000 }
gfCNCPoint5[14208] = {X 210.7271, Y 92.0536, Z -7.1667, A 0.000, B 0.000, C 0.000 }
gfCNCPoint5[14209] = {X 211.1032, Y 92.3082, Z -7.1667, A 0.000, B 0.000, C 0.000 }
gfCNCPoint5[14210] = {X 211.5318, Y 92.4581, Z -7.1667, A 0.000, B 0.000, C 0.000 }
gfCNCPoint5[14211] = {X 212.1208, Y 92.5821, Z -7.1667, A 0.000, B 0.000, C 0.000 }
gfCNCPoint5[14212] = {X 213.3773, Y 92.7403, Z -7.1667, A 0.000, B 0.000, C 0.000 }
gfCNCPoint5[14213] = {X 213.3917, Y 92.7388, Z -7.1667, A 0.000, B 0.000, C 0.000 }
gfCNCPoint5[14214] = {X 214.4501, Y 92.6555, Z -7.1667, A 0.000, B 0.000, C 0.000 }
gfCNCPoint5[14215] = {X 215.5101, Y 92.5945, Z -7.1667, A 0.000, B 0.000, C 0.000 }
gfCNCPoint5[14216] = {X 216.1641, Y 92.5226, Z -7.1667, A 0.000, B 0.000, C 0.000 }
gfCNCPoint5[14217] = {X 216.7938, Y 92.3319, Z -7.1667, A 0.000, B 0.000, C 0.000 }
gfCNCPoint5[14218] = {X 217.3777, Y 92.0288, Z -7.1667, A 0.000, B 0.000, C 0.000 }
gfCNCPoint5[14219] = {X 222.9188, Y 88.4528, Z -7.1667, A 0.000, B 0.000, C 0.000 }
gfCNCPoint5[14220] = {X 245.6518, Y 73.9168, Z -7.1667, A 0.000, B 0.000, C 0.000 }
gfCNCPoint5[14221] = {X 221.6009, Y 64.4790, Z -7.1667, A 0.000, B 0.000, C 0.000 }
gfCNCPoint5[14222] = {X 219.8422, Y 63.8905, Z -7.1667, A 0.000, B 0.000, C 0.000 }
gfCNCPoint5[14223] = {X 218.0278, Y 63.5063, Z -7.1667, A 0.000, B 0.000, C 0.000 }
gfCNCPoint5[14224] = {X 216.1815, Y 63.3315, Z -7.1667, A 0.000, B 0.000, C 0.000 }
gfCNCPoint5[14225] = {X 215.2274, Y 63.1935, Z -7.1667, A 0.000, B 0.000, C 0.000 }
gfCNCPoint5[14226] = {X 214.3262, Y 62.8509, Z -7.1667, A 0.000, B 0.000, C 0.000 }
gfCNCPoint5[14227] = {X 213.5213, Y 62.3203, Z -7.1667, A 0.000, B 0.000, C 0.000 }
gfCNCPoint5[14228] = {X 212.8512, Y 61.6271, Z -7.1667, A 0.000, B 0.000, C 0.000 }
gfCNCPoint5[14229] = {X 212.3482, Y 60.8046, Z -7.1667, A 0.000, B 0.000, C 0.000 }
gfCNCPoint5[14230] = {X 212.0364, Y 59.8923, Z -7.1667, A 0.000, B 0.000, C 0.000 }
gfCNCPoint5[14231] = {X 211.9308, Y 58.9341, Z -7.1667, A 0.000, B 0.000, C 0.000 }
gfCNCPoint5[14232] = {X 211.9308, Y 58.0000, Z -7.1667, A 0.000, B 0.000, C 0.000 }
gfCNCPoint5[14233] = {X 212.0411, Y 57.0209, Z -7.1667, A 0.000, B 0.000, C 0.000 }
gfCNCPoint5[14234] = {X 212.3665, Y 56.0909, Z -7.1667, A 0.000, B 0.000, C 0.000 }
gfCNCPoint5[14235] = {X 212.8907, Y 55.2566, Z -7.1667, A 0.000, B 0.000, C 0.000 }
gfCNCPoint5[14236] = {X 213.5875, Y 54.5599, Z -7.1667, A 0.000, B 0.000, C 0.000 }
gfCNCPoint5[14237] = {X 214.4217, Y 54.0357, Z -7.1667, A 0.000, B 0.000, C 0.000 }
gfCNCPoint5[14238] = {X 215.3517, Y 53.7103, Z -7.1667, A 0.000, B 0.000, C 0.000 }
gfCNCPoint5[14239] = {X 216.3308, Y 53.6000, Z -7.1667, A 0.000, B 0.000, C 0.000 }
gfCNCPoint5[14240] = {X 237.2617, Y 53.6000, Z -7.1667, A 0.000, B 0.000, C 0.000 }
gfCNCPoint5[14241] = {X 238.2408, Y 53.7103, Z -7.1667, A 0.000, B 0.000, C 0.000 }
gfCNCPoint5[14242] = {X 239.1708, Y 54.0357, Z -7.1667, A 0.000, B 0.000, C 0.000 }
gfCNCPoint5[14243] = {X 240.0050, Y 54.5599, Z -7.1667, A 0.000, B 0.000, C 0.000 }
gfCNCPoint5[14244] = {X 240.7017, Y 55.2566, Z -7.1667, A 0.000, B 0.000, C 0.000 }
gfCNCPoint5[14245] = {X 241.2260, Y 56.0909, Z -7.1667, A 0.000, B 0.000, C 0.000 }
gfCNCPoint5[14246] = {X 241.5514, Y 57.0209, Z -7.1667, A 0.000, B 0.000, C 0.000 }
gfCNCPoint5[14247] = {X 241.6617, Y 58.0000, Z -7.1667, A 0.000, B 0.000, C 0.000 }
gfCNCPoint5[14248] = {X 241.6617, Y 58.1771, Z -7.1667, A 0.000, B 0.000, C 0.000 }
gfCNCPoint5[14249] = {X 248.1452, Y 60.7053, Z -7.1667, A 0.000, B 0.000, C 0.000 }
gfCNCPoint5[14250] = {X 275.5518, Y 71.5835, Z -7.1667, A 0.000, B 0.000, C 0.000 }
gfCNCPoint5[14251] = {X 275.5515, Y 63.2810, Z -7.1667, A 0.000, B 0.000, C 0.000 }
gfCNCPoint5[14252] = {X 274.6925, Y 63.0557, Z -7.1667, A 0.000, B 0.000, C 0.000 }
gfCNCPoint5[14253] = {X 273.8961, Y 62.6624, Z -7.1667, A 0.000, B 0.000, C 0.000 }
gfCNCPoint5[14254] = {X 273.1950, Y 62.1172, Z -7.1667, A 0.000, B 0.000, C 0.000 }
gfCNCPoint5[14255] = {X 272.6177, Y 61.4423, Z -7.1667, A 0.000, B 0.000, C 0.000 }
gfCNCPoint5[14256] = {X 272.1876, Y 60.6653, Z -7.1667, A 0.000, B 0.000, C 0.000 }
gfCNCPoint5[14257] = {X 271.9223, Y 59.8177, Z -7.1667, A 0.000, B 0.000, C 0.000 }
gfCNCPoint5[14258] = {X 271.8327, Y 58.9341, Z -7.1667, A 0.000, B 0.000, C 0.000 }
gfCNCPoint5[14259] = {X 271.8327, Y 58.0000, Z -7.1667, A 0.000, B 0.000, C 0.000 }
gfCNCPoint5[14260] = {X 271.9430, Y 57.0209, Z -7.1667, A 0.000, B 0.000, C 0.000 }
gfCNCPoint5[14261] = {X 272.2684, Y 56.0909, Z -7.1667, A 0.000, B 0.000, C 0.000 }
gfCNCPoint5[14262] = {X 272.7926, Y 55.2566, Z -7.1667, A 0.000, B 0.000, C 0.000 }
gfCNCPoint5[14263] = {X 273.4893, Y 54.5599, Z -7.1667, A 0.000, B 0.000, C 0.000 }
gfCNCPoint5[14264] = {X 274.3236, Y 54.0357, Z -7.1667, A 0.000, B 0.000, C 0.000 }
gfCNCPoint5[14265] = {X 275.2536, Y 53.7103, Z -7.1667, A 0.000, B 0.000, C 0.000 }
gfCNCPoint5[14266] = {X 276.2327, Y 53.6000, Z -7.1667, A 0.000, B 0.000, C 0.000 }
gfCNCPoint5[14267] = {X 292.7731, Y 53.6000, Z -7.1667, A 0.000, B 0.000, C 0.000 }
gfCNCPoint5[14268] = {X 293.7522, Y 53.7103, Z -7.1667, A 0.000, B 0.000, C 0.000 }
gfCNCPoint5[14269] = {X 294.6822, Y 54.0357, Z -7.1667, A 0.000, B 0.000, C 0.000 }
gfCNCPoint5[14270] = {X 295.5164, Y 54.5599, Z -7.1667, A 0.000, B 0.000, C 0.000 }
gfCNCPoint5[14271] = {X 296.2131, Y 55.2566, Z -7.1667, A 0.000, B 0.000, C 0.000 }
gfCNCPoint5[14272] = {X 296.7373, Y 56.0909, Z -7.1667, A 0.000, B 0.000, C 0.000 }
gfCNCPoint5[14273] = {X 297.0628, Y 57.0209, Z -7.1667, A 0.000, B 0.000, C 0.000 }
gfCNCPoint5[14274] = {X 297.1731, Y 58.0000, Z -7.1667, A 0.000, B 0.000, C 0.000 }
gfCNCPoint5[14275] = {X 297.1731, Y 58.9352, Z -7.1667, A 0.000, B 0.000, C 0.000 }
gfCNCPoint5[14276] = {X 297.0814, Y 59.8182, Z -7.1667, A 0.000, B 0.000, C 0.000 }
gfCNCPoint5[14277] = {X 296.8150, Y 60.6651, Z -7.1667, A 0.000, B 0.000, C 0.000 }
gfCNCPoint5[14278] = {X 296.3845, Y 61.4415, Z -7.1667, A 0.000, B 0.000, C 0.000 }
gfCNCPoint5[14279] = {X 295.8075, Y 62.1162, Z -7.1667, A 0.000, B 0.000, C 0.000 }
gfCNCPoint5[14280] = {X 295.1072, Y 62.6618, Z -7.1667, A 0.000, B 0.000, C 0.000 }
gfCNCPoint5[14281] = {X 294.3119, Y 63.0563, Z -7.1667, A 0.000, B 0.000, C 0.000 }
gfCNCPoint5[14282] = {X 293.4538, Y 63.2838, Z -7.1667, A 0.000, B 0.000, C 0.000 }
gfCNCPoint5[14283] = {X 293.4538, Y 92.7100, Z -7.1667, A 0.000, B 0.000, C 0.000 }
gfCNCPoint5[14284] = {X 294.3116, Y 92.9399, Z -7.1667, A 0.000, B 0.000, C 0.000 }
gfCNCPoint5[14285] = {X 295.1064, Y 93.3364, Z -7.1667, A 0.000, B 0.000, C 0.000 }
gfCNCPoint5[14286] = {X 295.8062, Y 93.8833, Z -7.1667, A 0.000, B 0.000, C 0.000 }
gfCNCPoint5[14287] = {X 296.3830, Y 94.5587, Z -7.1667, A 0.000, B 0.000, C 0.000 }
gfCNCPoint5[14288] = {X 296.8134, Y 95.3356, Z -7.1667, A 0.000, B 0.000, C 0.000 }
gfCNCPoint5[14289] = {X 297.0804, Y 96.1827, Z -7.1667, A 0.000, B 0.000, C 0.000 }
gfCNCPoint5[14290] = {X 297.1731, Y 97.0660, Z -7.1667, A 0.000, B 0.000, C 0.000 }
gfCNCPoint5[14291] = {X 297.1731, Y 97.6951, Z -7.1667, A 0.000, B 0.000, C 0.000 }
gfCNCPoint5[14292] = {X 297.6531, Y 97.6951, Z -7.1667, A 0.000, B 0.000, C 0.000 }
gfCNCPoint5[14293] = {X 314.2118, Y 97.6951, Z -7.1667, A 0.000, B 0.000, C 0.000 }
gfCNCPoint5[14294] = {X 313.0146, Y 96.8450, Z -7.1667, A 0.000, B 0.000, C 0.000 }
gfCNCPoint5[14295] = {X 311.8813, Y 95.9112, Z -7.1667, A 0.000, B 0.000, C 0.000 }
gfCNCPoint5[14296] = {X 310.9057, Y 94.9490, Z -7.1667, A 0.000, B 0.000, C 0.000 }
gfCNCPoint5[14297] = {X 310.0413, Y 93.8857, Z -7.1667, A 0.000, B 0.000, C 0.000 }
gfCNCPoint5[14298] = {X 309.2072, Y 92.5710, Z -7.1667, A 0.000, B 0.000, C 0.000 }
gfCNCPoint5[14299] = {X 308.5432, Y 91.1627, Z -7.1667, A 0.000, B 0.000, C 0.000 }
gfCNCPoint5[14300] = {X 308.0596, Y 89.6828, Z -7.1667, A 0.000, B 0.000, C 0.000 }
gfCNCPoint5[14301] = {X 307.7061, Y 88.0129, Z -7.1667, A 0.000, B 0.000, C 0.000 }
gfCNCPoint5[14302] = {X 307.4972, Y 86.3188, Z -7.1667, A 0.000, B 0.000, C 0.000 }
gfCNCPoint5[14303] = {X 307.4344, Y 84.6131, Z -7.1667, A 0.000, B 0.000, C 0.000 }
gfCNCPoint5[14304] = {X 307.4356, Y 63.6740, Z -7.1667, A 0.000, B 0.000, C 0.000 }
gfCNCPoint5[14305] = {X 306.4274, Y 63.3056, Z -7.1667, A 0.000, B 0.000, C 0.000 }
gfCNCPoint5[14306] = {X 305.5242, Y 62.7257, Z -7.1667, A 0.000, B 0.000, C 0.000 }
gfCNCPoint5[14307] = {X 304.7695, Y 61.9624, Z -7.1667, A 0.000, B 0.000, C 0.000 }
gfCNCPoint5[14308] = {X 304.2000, Y 61.0526, Z -7.1667, A 0.000, B 0.000, C 0.000 }
gfCNCPoint5[14309] = {X 303.8432, Y 60.0402, Z -7.1667, A 0.000, B 0.000, C 0.000 }
gfCNCPoint5[14310] = {X 303.7164, Y 58.9744, Z -7.1667, A 0.000, B 0.000, C 0.000 }
gfCNCPoint5[14311] = {X 303.7162, Y 58.0000, Z -7.1667, A 0.000, B 0.000, C 0.000 }
gfCNCPoint5[14312] = {X 303.8100, Y 57.0480, Z -7.1667, A 0.000, B 0.000, C 0.000 }
gfCNCPoint5[14313] = {X 304.0877, Y 56.1325, Z -7.1667, A 0.000, B 0.000, C 0.000 }
gfCNCPoint5[14314] = {X 304.5387, Y 55.2888, Z -7.1667, A 0.000, B 0.000, C 0.000 }
gfCNCPoint5[14315] = {X 305.1455, Y 54.5493, Z -7.1667, A 0.000, B 0.000, C 0.000 }
gfCNCPoint5[14316] = {X 305.8850, Y 53.9424, Z -7.1667, A 0.000, B 0.000, C 0.000 }
gfCNCPoint5[14317] = {X 306.7287, Y 53.4915, Z -7.1667, A 0.000, B 0.000, C 0.000 }
gfCNCPoint5[14318] = {X 307.6442, Y 53.2138, Z -7.1667, A 0.000, B 0.000, C 0.000 }
gfCNCPoint5[14319] = {X 308.5962, Y 53.1200, Z -7.1667, A 0.000, B 0.000, C 0.000 }
gfCNCPoint5[14320] = {X 324.3107, Y 53.1200, Z -7.1667, A 0.000, B 0.000, C 0.000 }
gfCNCPoint5[14321] = {X 325.2627, Y 53.2138, Z -7.1667, A 0.000, B 0.000, C 0.000 }
gfCNCPoint5[14322] = {X 326.1782, Y 53.4915, Z -7.1667, A 0.000, B 0.000, C 0.000 }
gfCNCPoint5[14323] = {X 327.0219, Y 53.9424, Z -7.1667, A 0.000, B 0.000, C 0.000 }
gfCNCPoint5[14324] = {X 327.7614, Y 54.5493, Z -7.1667, A 0.000, B 0.000, C 0.000 }
gfCNCPoint5[14325] = {X 328.3683, Y 55.2888, Z -7.1667, A 0.000, B 0.000, C 0.000 }
gfCNCPoint5[14326] = {X 328.8192, Y 56.1325, Z -7.1667, A 0.000, B 0.000, C 0.000 }
gfCNCPoint5[14327] = {X 329.0969, Y 57.0480, Z -7.1667, A 0.000, B 0.000, C 0.000 }
gfCNCPoint5[14328] = {X 329.1907, Y 58.0000, Z -7.1667, A 0.000, B 0.000, C 0.000 }
gfCNCPoint5[14329] = {X 329.1907, Y 58.9341, Z -7.1667, A 0.000, B 0.000, C 0.000 }
gfCNCPoint5[14330] = {X 329.0675, Y 60.0068, Z -7.1667, A 0.000, B 0.000, C 0.000 }
gfCNCPoint5[14331] = {X 328.7131, Y 61.0268, Z -7.1667, A 0.000, B 0.000, C 0.000 }
gfCNCPoint5[14332] = {X 328.1447, Y 61.9448, Z -7.1667, A 0.000, B 0.000, C 0.000 }
gfCNCPoint5[14333] = {X 327.3896, Y 62.7166, Z -7.1667, A 0.000, B 0.000, C 0.000 }
gfCNCPoint5[14334] = {X 326.4843, Y 63.3051, Z -7.1667, A 0.000, B 0.000, C 0.000 }
gfCNCPoint5[14335] = {X 325.4724, Y 63.6817, Z -7.1667, A 0.000, B 0.000, C 0.000 }
gfCNCPoint5[14336] = {X 325.4742, Y 83.2269, Z -7.1667, A 0.000, B 0.000, C 0.000 }
gfCNCPoint5[14337] = {X 325.4877, Y 84.6073, Z -7.1667, A 0.000, B 0.000, C 0.000 }
gfCNCPoint5[14338] = {X 325.5521, Y 85.7050, Z -7.1667, A 0.000, B 0.000, C 0.000 }
gfCNCPoint5[14339] = {X 325.7362, Y 86.7890, Z -7.1667, A 0.000, B 0.000, C 0.000 }
gfCNCPoint5[14340] = {X 326.0551, Y 87.0640, Z -7.1667, A 0.000, B 0.000, C 0.000 }
gfCNCPoint5[14341] = {X 326.4234, Y 87.2684, Z -7.1667, A 0.000, B 0.000, C 0.000 }
gfCNCPoint5[14342] = {X 328.1519, Y 87.9618, Z -7.1667, A 0.000, B 0.000, C 0.000 }
gfCNCPoint5[14343] = {X 329.9516, Y 88.4412, Z -7.1667, A 0.000, B 0.000, C 0.000 }
gfCNCPoint5[14344] = {X 333.0038, Y 88.9890, Z -7.1667, A 0.000, B 0.000, C 0.000 }
gfCNCPoint5[14345] = {X 336.0838, Y 89.3497, Z -7.1667, A 0.000, B 0.000, C 0.000 }
gfCNCPoint5[14346] = {X 340.4352, Y 89.6427, Z -7.1667, A 0.000, B 0.000, C 0.000 }
gfCNCPoint5[14347] = {X 344.7937, Y 89.7958, Z -7.1667, A 0.000, B 0.000, C 0.000 }
gfCNCPoint5[14348] = {X 349.1549, Y 89.8091, Z -7.1667, A 0.000, B 0.000, C 0.000 }
gfCNCPoint5[14349] = {X 353.2889, Y 89.7413, Z -7.1667, A 0.000, B 0.000, C 0.000 }
gfCNCPoint5[14350] = {X 357.4177, Y 89.5234, Z -7.1667, A 0.000, B 0.000, C 0.000 }
gfCNCPoint5[14351] = {X 361.5359, Y 89.1556, Z -7.1667, A 0.000, B 0.000, C 0.000 }
gfCNCPoint5[14352] = {X 363.5861, Y 88.8728, Z -7.1667, A 0.000, B 0.000, C 0.000 }
gfCNCPoint5[14353] = {X 365.6175, Y 88.4768, Z -7.1667, A 0.000, B 0.000, C 0.000 }
gfCNCPoint5[14354] = {X 367.6239, Y 87.9688, Z -7.1667, A 0.000, B 0.000, C 0.000 }
gfCNCPoint5[14355] = {X 368.9176, Y 87.4945, Z -7.1667, A 0.000, B 0.000, C 0.000 }
gfCNCPoint5[14356] = {X 370.1130, Y 86.8094, Z -7.1667, A 0.000, B 0.000, C 0.000 }
gfCNCPoint5[14357] = {X 370.2975, Y 85.3242, Z -7.1667, A 0.000, B 0.000, C 0.000 }
gfCNCPoint5[14358] = {X 370.3591, Y 83.8289, Z -7.1667, A 0.000, B 0.000, C 0.000 }
gfCNCPoint5[14359] = {X 370.3579, Y 63.6739, Z -7.1667, A 0.000, B 0.000, C 0.000 }
gfCNCPoint5[14360] = {X 369.3499, Y 63.3054, Z -7.1667, A 0.000, B 0.000, C 0.000 }
gfCNCPoint5[14361] = {X 368.4468, Y 62.7254, Z -7.1667, A 0.000, B 0.000, C 0.000 }
gfCNCPoint5[14362] = {X 367.6924, Y 61.9621, Z -7.1667, A 0.000, B 0.000, C 0.000 }
gfCNCPoint5[14363] = {X 367.1230, Y 61.0523, Z -7.1667, A 0.000, B 0.000, C 0.000 }
gfCNCPoint5[14364] = {X 366.7663, Y 60.0401, Z -7.1667, A 0.000, B 0.000, C 0.000 }
gfCNCPoint5[14365] = {X 366.6394, Y 58.9744, Z -7.1667, A 0.000, B 0.000, C 0.000 }
gfCNCPoint5[14366] = {X 366.6393, Y 58.0000, Z -7.1667, A 0.000, B 0.000, C 0.000 }
gfCNCPoint5[14367] = {X 366.7331, Y 57.0480, Z -7.1667, A 0.000, B 0.000, C 0.000 }
gfCNCPoint5[14368] = {X 367.0108, Y 56.1325, Z -7.1667, A 0.000, B 0.000, C 0.000 }
gfCNCPoint5[14369] = {X 367.4617, Y 55.2888, Z -7.1667, A 0.000, B 0.000, C 0.000 }
gfCNCPoint5[14370] = {X 368.0686, Y 54.5493, Z -7.1667, A 0.000, B 0.000, C 0.000 }
gfCNCPoint5[14371] = {X 368.8081, Y 53.9424, Z -7.1667, A 0.000, B 0.000, C 0.000 }
gfCNCPoint5[14372] = {X 369.6518, Y 53.4915, Z -7.1667, A 0.000, B 0.000, C 0.000 }
gfCNCPoint5[14373] = {X 370.5672, Y 53.2138, Z -7.1667, A 0.000, B 0.000, C 0.000 }
gfCNCPoint5[14374] = {X 371.5193, Y 53.1200, Z -7.1667, A 0.000, B 0.000, C 0.000 }
gfCNCPoint5[14375] = {X 388.0597, Y 53.1200, Z -7.1667, A 0.000, B 0.000, C 0.000 }
gfCNCPoint5[14376] = {X 389.0355, Y 53.2186, Z -7.1667, A 0.000, B 0.000, C 0.000 }
gfCNCPoint5[14377] = {X 389.9719, Y 53.5102, Z -7.1667, A 0.000, B 0.000, C 0.000 }
gfCNCPoint5[14378] = {X 390.8310, Y 53.9833, Z -7.1667, A 0.000, B 0.000, C 0.000 }
gfCNCPoint5[14379] = {X 391.5783, Y 54.6186, Z -7.1667, A 0.000, B 0.000, C 0.000 }
gfCNCPoint5[14380] = {X 392.1572, Y 55.3496, Z -7.1667, A 0.000, B 0.000, C 0.000 }
gfCNCPoint5[14381] = {X 392.5865, Y 56.1774, Z -7.1667, A 0.000, B 0.000, C 0.000 }
gfCNCPoint5[14382] = {X 392.8506, Y 57.0718, Z -7.1667, A 0.000, B 0.000, C 0.000 }
gfCNCPoint5[14383] = {X 392.9397, Y 58.0000, Z -7.1667, A 0.000, B 0.000, C 0.000 }
gfCNCPoint5[14384] = {X 392.9395, Y 58.9743, Z -7.1667, A 0.000, B 0.000, C 0.000 }
gfCNCPoint5[14385] = {X 392.8794, Y 59.6988, Z -7.1667, A 0.000, B 0.000, C 0.000 }
gfCNCPoint5[14386] = {X 392.7123, Y 60.4064, Z -7.1667, A 0.000, B 0.000, C 0.000 }
gfCNCPoint5[14387] = {X 392.4419, Y 61.0813, Z -7.1667, A 0.000, B 0.000, C 0.000 }
gfCNCPoint5[14388] = {X 392.0575, Y 61.7331, Z -7.1667, A 0.000, B 0.000, C 0.000 }
gfCNCPoint5[14389] = {X 391.5774, Y 62.3180, Z -7.1667, A 0.000, B 0.000, C 0.000 }
gfCNCPoint5[14390] = {X 390.8821, Y 62.9185, Z -7.1667, A 0.000, B 0.000, C 0.000 }
gfCNCPoint5[14391] = {X 390.0870, Y 63.3789, Z -7.1667, A 0.000, B 0.000, C 0.000 }
gfCNCPoint5[14392] = {X 389.2200, Y 63.6828, Z -7.1667, A 0.000, B 0.000, C 0.000 }
gfCNCPoint5[14393] = {X 389.2179, Y 84.6139, Z -7.1667, A 0.000, B 0.000, C 0.000 }
gfCNCPoint5[14394] = {X 389.1561, Y 86.3199, Z -7.1667, A 0.000, B 0.000, C 0.000 }
gfCNCPoint5[14395] = {X 388.9457, Y 88.0141, Z -7.1667, A 0.000, B 0.000, C 0.000 }
gfCNCPoint5[14396] = {X 388.5885, Y 89.6835, Z -7.1667, A 0.000, B 0.000, C 0.000 }
gfCNCPoint5[14397] = {X 388.1049, Y 91.1631, Z -7.1667, A 0.000, B 0.000, C 0.000 }
gfCNCPoint5[14398] = {X 387.4409, Y 92.5709, Z -7.1667, A 0.000, B 0.000, C 0.000 }
gfCNCPoint5[14399] = {X 386.6067, Y 93.8852, Z -7.1667, A 0.000, B 0.000, C 0.000 }
gfCNCPoint5[14400] = {X 385.8750, Y 94.7997, Z -7.1667, A 0.000, B 0.000, C 0.000 }
gfCNCPoint5[14401] = {X 385.0607, Y 95.6415, Z -7.1667, A 0.000, B 0.000, C 0.000 }
gfCNCPoint5[14402] = {X 383.8009, Y 96.7249, Z -7.1667, A 0.000, B 0.000, C 0.000 }
gfCNCPoint5[14403] = {X 382.4521, Y 97.6951, Z -7.1667, A 0.000, B 0.000, C 0.000 }
gfCNCPoint5[14404] = {X 382.1889, Y 97.2937, Z -7.1667, A 0.000, B 0.000, C 0.000 }
gfCNCPoint5[14405] = {X 381.0205, Y 98.0000, Z -7.1667, A 0.000, B 0.000, C 0.000 }
gfCNCPoint5[14406] = {X 379.8038, Y 98.6193, Z -7.1667, A 0.000, B 0.000, C 0.000 }
gfCNCPoint5[14407] = {X 377.5265, Y 99.5766, Z -7.1667, A 0.000, B 0.000, C 0.000 }
gfCNCPoint5[14408] = {X 375.1866, Y 100.3688, Z -7.1667, A 0.000, B 0.000, C 0.000 }
gfCNCPoint5[14409] = {X 372.7961, Y 100.9917, Z -7.1667, A 0.000, B 0.000, C 0.000 }
gfCNCPoint5[14410] = {X 368.8818, Y 101.7455, Z -7.1667, A 0.000, B 0.000, C 0.000 }
gfCNCPoint5[14411] = {X 364.9352, Y 102.3063, Z -7.1667, A 0.000, B 0.000, C 0.000 }
gfCNCPoint5[14412] = {X 360.9659, Y 102.6726, Z -7.1667, A 0.000, B 0.000, C 0.000 }
gfCNCPoint5[14413] = {X 355.2456, Y 102.9777, Z -7.1667, A 0.000, B 0.000, C 0.000 }
gfCNCPoint5[14414] = {X 349.5186, Y 103.1078, Z -7.1667, A 0.000, B 0.000, C 0.000 }
gfCNCPoint5[14415] = {X 343.7903, Y 103.0628, Z -7.1667, A 0.000, B 0.000, C 0.000 }
gfCNCPoint5[14416] = {X 338.0660, Y 102.8427, Z -7.1667, A 0.000, B 0.000, C 0.000 }
gfCNCPoint5[14417] = {X 334.1085, Y 102.5655, Z -7.1667, A 0.000, B 0.000, C 0.000 }
gfCNCPoint5[14418] = {X 330.1659, Y 102.1233, Z -7.1667, A 0.000, B 0.000, C 0.000 }
gfCNCPoint5[14419] = {X 326.2453, Y 101.5168, Z -7.1667, A 0.000, B 0.000, C 0.000 }
gfCNCPoint5[14420] = {X 323.3901, Y 100.9107, Z -7.1667, A 0.000, B 0.000, C 0.000 }
gfCNCPoint5[14421] = {X 320.5872, Y 100.0962, Z -7.1667, A 0.000, B 0.000, C 0.000 }
gfCNCPoint5[14422] = {X 317.8519, Y 99.0776, Z -7.1667, A 0.000, B 0.000, C 0.000 }
gfCNCPoint5[14423] = {X 316.3330, Y 98.3769, Z -7.1667, A 0.000, B 0.000, C 0.000 }
gfCNCPoint5[14424] = {X 314.8779, Y 97.5518, Z -7.1667, A 0.000, B 0.000, C 0.000 }
gfCNCPoint5[14425] = {X 313.4969, Y 96.6079, Z -7.1667, A 0.000, B 0.000, C 0.000 }
gfCNCPoint5[14426] = {X 312.1996, Y 95.5520, Z -7.1667, A 0.000, B 0.000, C 0.000 }
gfCNCPoint5[14427] = {X 311.1891, Y 94.5464, Z -7.1667, A 0.000, B 0.000, C 0.000 }
gfCNCPoint5[14428] = {X 310.3047, Y 93.4281, Z -7.1667, A 0.000, B 0.000, C 0.000 }
gfCNCPoint5[14429] = {X 309.5591, Y 92.2130, Z -7.1667, A 0.000, B 0.000, C 0.000 }
gfCNCPoint5[14430] = {X 308.9628, Y 90.9181, Z -7.1667, A 0.000, B 0.000, C 0.000 }
gfCNCPoint5[14431] = {X 308.5240, Y 89.5616, Z -7.1667, A 0.000, B 0.000, C 0.000 }
gfCNCPoint5[14432] = {X 308.1792, Y 87.9321, Z -7.1667, A 0.000, B 0.000, C 0.000 }
gfCNCPoint5[14433] = {X 307.9755, Y 86.2791, Z -7.1667, A 0.000, B 0.000, C 0.000 }
gfCNCPoint5[14434] = {X 307.9144, Y 84.6146, Z -7.1667, A 0.000, B 0.000, C 0.000 }
gfCNCPoint5[14435] = {X 307.9156, Y 63.2811, Z -7.1667, A 0.000, B 0.000, C 0.000 }
gfCNCPoint5[14436] = {X 307.0564, Y 63.0558, Z -7.1667, A 0.000, B 0.000, C 0.000 }
gfCNCPoint5[14437] = {X 306.2600, Y 62.6626, Z -7.1667, A 0.000, B 0.000, C 0.000 }
gfCNCPoint5[14438] = {X 305.5588, Y 62.1174, Z -7.1667, A 0.000, B 0.000, C 0.000 }
gfCNCPoint5[14439] = {X 304.9813, Y 61.4425, Z -7.1667, A 0.000, B 0.000, C 0.000 }
gfCNCPoint5[14440] = {X 304.5512, Y 60.6654, Z -7.1667, A 0.000, B 0.000, C 0.000 }
gfCNCPoint5[14441] = {X 304.2859, Y 59.8177, Z -7.1667, A 0.000, B 0.000, C 0.000 }
gfCNCPoint5[14442] = {X 304.1962, Y 58.9341, Z -7.1667, A 0.000, B 0.000, C 0.000 }
gfCNCPoint5[14443] = {X 304.1962, Y 58.0000, Z -7.1667, A 0.000, B 0.000, C 0.000 }
gfCNCPoint5[14444] = {X 304.3065, Y 57.0209, Z -7.1667, A 0.000, B 0.000, C 0.000 }
gfCNCPoint5[14445] = {X 304.6320, Y 56.0909, Z -7.1667, A 0.000, B 0.000, C 0.000 }
gfCNCPoint5[14446] = {X 305.1562, Y 55.2566, Z -7.1667, A 0.000, B 0.000, C 0.000 }
gfCNCPoint5[14447] = {X 305.8529, Y 54.5599, Z -7.1667, A 0.000, B 0.000, C 0.000 }
